# B&R Automation Studio project Ampel (part 5)

```cpp
#if HFSM2_PLANS_AVAILABLE()
		HFSM2_CONSTEXPR(14)	TaskStatus	wideUpdatePlans		 ( FullControl& control												   )		noexcept;
#endif

		HFSM2_CONSTEXPR(14)	bool		wideForwardExitGuard (GuardControl& control,						const ProngCBits prongs)		noexcept;
		HFSM2_CONSTEXPR(14)	bool		wideForwardExitGuard (GuardControl& control												   )		noexcept;
		HFSM2_CONSTEXPR(14)	bool		wideExitGuard		 (GuardControl& control												   )		noexcept;

		HFSM2_CONSTEXPR(14)	void		wideExit			 ( PlanControl& control												   )		noexcept;

		HFSM2_CONSTEXPR(14)	void		wideForwardActive	 (	   Control& control, const Request request, const ProngCBits prongs)		noexcept;
		HFSM2_CONSTEXPR(14)	void		wideForwardRequest	 (	   Control& control, const Request request						   )		noexcept;

		HFSM2_CONSTEXPR(14)	void		wideRequestChange	 (	   Control& control, const Request request						   )		noexcept;
		HFSM2_CONSTEXPR(14)	void		wideRequestRestart	 (	   Control& control, const Request request						   )		noexcept;
		HFSM2_CONSTEXPR(14)	void		wideRequestResume	 (	   Control& control, const Request request						   )		noexcept;
		HFSM2_CONSTEXPR(14)	void		wideRequestSelect	 (	   Control& control, const Request request						   )		noexcept;

#if HFSM2_UTILITY_THEORY_AVAILABLE()
		HFSM2_CONSTEXPR(14)	void		wideRequestUtilize	 (	   Control& control, const Request request						   )		noexcept;
		HFSM2_CONSTEXPR(14)	void		wideRequestRandomize (	   Control& control, const Request request						   )		noexcept;

		HFSM2_CONSTEXPR(14)	Utility		wideReportChange	 (	   Control& control												   )		noexcept;
		HFSM2_CONSTEXPR(14)	Utility		wideReportUtilize	 (	   Control& control												   )		noexcept;
		HFSM2_CONSTEXPR(14)	Utility		wideReportRandomize  (	   Control& control												   )		noexcept;
#endif

		HFSM2_CONSTEXPR(14)	void		wideChangeToRequested( PlanControl& control												   )		noexcept;

#if HFSM2_SERIALIZATION_AVAILABLE()
		using WriteStream	= typename Args::WriteStream;
		using ReadStream	= typename Args::ReadStream;

		HFSM2_CONSTEXPR(14)	void		wideSaveActive		  (const Registry& registry, WriteStream& stream)  const noexcept;
		HFSM2_CONSTEXPR(14)	void		wideSaveResumable	  (const Registry& registry, WriteStream& stream)  const noexcept;

		HFSM2_CONSTEXPR(14)	void		wideLoadRequested	  (		 Registry& registry,  ReadStream& stream)  const noexcept;
		HFSM2_CONSTEXPR(14)	void		wideLoadResumable	  (		 Registry& registry,  ReadStream& stream)  const noexcept;
#endif

#if HFSM2_STRUCTURE_REPORT_AVAILABLE()
		using StructureStateInfos = typename Args::StructureStateInfos;

		static constexpr Long NAME_COUNT	 = Initial::NAME_COUNT  + Remaining::NAME_COUNT;

		HFSM2_CONSTEXPR(14)	void wideGetNames(const Long parent,
		const Short depth,
		StructureStateInfos& stateInfos)	  const noexcept;
#endif

	};

}
}

namespace hfsm2 {
	namespace detail {

		template <typename TN_, typename TA_, Prong NP_, typename TI_, typename... TR_>
		HFSM2_CONSTEXPR(14)
		void
		OS_<TN_, TA_, NP_, TI_, TR_...>::wideRegister(Registry& registry,
		const ForkID forkId) noexcept
		{
		Initial	 ::deepRegister(registry, Parent{forkId, PRONG_INDEX});
		Remaining::wideRegister(registry,		 forkId				 );
	}

	template <typename TN_, typename TA_, Prong NP_, typename TI_, typename... TR_>
	HFSM2_CONSTEXPR(14)
	bool
	OS_<TN_, TA_, NP_, TI_, TR_...>::wideForwardEntryGuard(GuardControl& control,
	const ProngCBits prongs) noexcept
	{
	const bool i = prongs.get(PRONG_INDEX) ?
		Initial	::deepForwardEntryGuard(control		   ) : false;

	const bool r = Remaining::wideForwardEntryGuard(control, prongs);

	return i || r;
}

template <typename TN_, typename TA_, Prong NP_, typename TI_, typename... TR_>
HFSM2_CONSTEXPR(14)
bool
OS_<TN_, TA_, NP_, TI_, TR_...>::wideForwardEntryGuard(GuardControl& control) noexcept {
const bool i = Initial	::deepForwardEntryGuard(control);
const bool r = Remaining::wideForwardEntryGuard(control);

return i || r;
}

template <typename TN_, typename TA_, Prong NP_, typename TI_, typename... TR_>
HFSM2_CONSTEXPR(14)
bool
OS_<TN_, TA_, NP_, TI_, TR_...>::wideEntryGuard(GuardControl& control) noexcept {
const bool i = Initial	::deepEntryGuard(control);
const bool r = Remaining::wideEntryGuard(control);

return i || r;
}

template <typename TN_, typename TA_, Prong NP_, typename TI_, typename... TR_>
HFSM2_CONSTEXPR(14)
void
OS_<TN_, TA_, NP_, TI_, TR_...>::wideEnter(PlanControl& control) noexcept {
	Initial	 ::deepEnter(control);
	Remaining::wideEnter(control);
}

template <typename TN_, typename TA_, Prong NP_, typename TI_, typename... TR_>
HFSM2_CONSTEXPR(14)
void
OS_<TN_, TA_, NP_, TI_, TR_...>::wideReenter(PlanControl& control) noexcept {
	Initial	 ::deepReenter(control);
	Remaining::wideReenter(control);
}

template <typename TN_, typename TA_, Prong NP_, typename TI_, typename... TR_>
HFSM2_CONSTEXPR(14)
TaskStatus
OS_<TN_, TA_, NP_, TI_, TR_...>::widePreUpdate(FullControl& control) noexcept {
TaskStatus status;
	status |= Initial  ::deepPreUpdate(control);
	status |= Remaining::widePreUpdate(control);

return status;
}

template <typename TN_, typename TA_, Prong NP_, typename TI_, typename... TR_>
HFSM2_CONSTEXPR(14)
TaskStatus
OS_<TN_, TA_, NP_, TI_, TR_...>::wideUpdate(FullControl& control) noexcept {
TaskStatus status;
	status |= Initial  ::deepUpdate(control);
	status |= Remaining::wideUpdate(control);

return status;
}

template <typename TN_, typename TA_, Prong NP_, typename TI_, typename... TR_>
HFSM2_CONSTEXPR(14)
TaskStatus
OS_<TN_, TA_, NP_, TI_, TR_...>::widePostUpdate(FullControl& control) noexcept {
TaskStatus status;
	status |= Initial  ::deepPostUpdate(control);
	status |= Remaining::widePostUpdate(control);

return status;
}

template <typename TN_, typename TA_, Prong NP_, typename TI_, typename... TR_>
template <typename TEvent>
HFSM2_CONSTEXPR(14)
TaskStatus
OS_<TN_, TA_, NP_, TI_, TR_...>::widePreReact(EventControl& control,
											  const TEvent& event) noexcept
{
TaskStatus status;
	status |= Initial  ::deepPreReact(control, event);
	status |= Remaining::widePreReact(control, event);

return status;
}

template <typename TN_, typename TA_, Prong NP_, typename TI_, typename... TR_>
template <typename TEvent>
HFSM2_CONSTEXPR(14)
TaskStatus
OS_<TN_, TA_, NP_, TI_, TR_...>::wideReact(EventControl& control,
										   const TEvent& event) noexcept
{
TaskStatus status;
	status |= Initial  ::deepReact(control, event);
	status |= Remaining::wideReact(control, event);

return status;
}

template <typename TN_, typename TA_, Prong NP_, typename TI_, typename... TR_>
template <typename TEvent>
HFSM2_CONSTEXPR(14)
TaskStatus
OS_<TN_, TA_, NP_, TI_, TR_...>::widePostReact(EventControl& control,
											   const TEvent& event) noexcept
{
TaskStatus status;
	status |= Initial  ::deepPostReact(control, event);
	status |= Remaining::widePostReact(control, event);

return status;
}

template <typename TN_, typename TA_, Prong NP_, typename TI_, typename... TR_>
template <typename TEvent>
HFSM2_CONSTEXPR(14)
void
OS_<TN_, TA_, NP_, TI_, TR_...>::wideQuery(ConstControl& control,
										   TEvent& event) const noexcept
{
	Initial  ::deepQuery(control, event);
	Remaining::wideQuery(control, event);
}

#if HFSM2_PLANS_AVAILABLE()

template <typename TN_, typename TA_, Prong NP_, typename TI_, typename... TR_>
HFSM2_CONSTEXPR(14)
TaskStatus
OS_<TN_, TA_, NP_, TI_, TR_...>::wideUpdatePlans(FullControl& control) noexcept {
TaskStatus status;
	status |= Initial  ::deepUpdatePlans(control);
	status |= Remaining::wideUpdatePlans(control);

return status;
}

#endif

template <typename TN_, typename TA_, Prong NP_, typename TI_, typename... TR_>
HFSM2_CONSTEXPR(14)
bool
OS_<TN_, TA_, NP_, TI_, TR_...>::wideForwardExitGuard(GuardControl& control,
													  const ProngCBits prongs) noexcept
{
const bool i = prongs.get(PRONG_INDEX) ?
	Initial	::deepForwardExitGuard(control		  ) : false;

const bool r = Remaining::wideForwardExitGuard(control, prongs);

return i || r;
}

template <typename TN_, typename TA_, Prong NP_, typename TI_, typename... TR_>
HFSM2_CONSTEXPR(14)
bool
OS_<TN_, TA_, NP_, TI_, TR_...>::wideForwardExitGuard(GuardControl& control) noexcept {
const bool i = Initial	::deepForwardExitGuard(control);
const bool r = Remaining::wideForwardExitGuard(control);

return i || r;
}

template <typename TN_, typename TA_, Prong NP_, typename TI_, typename... TR_>
HFSM2_CONSTEXPR(14)
bool
OS_<TN_, TA_, NP_, TI_, TR_...>::wideExitGuard(GuardControl& control) noexcept {
const bool i = Initial	::deepExitGuard(control);
const bool r = Remaining::wideExitGuard(control);

return i || r;
}

template <typename TN_, typename TA_, Prong NP_, typename TI_, typename... TR_>
HFSM2_CONSTEXPR(14)
void
OS_<TN_, TA_, NP_, TI_, TR_...>::wideExit(PlanControl& control) noexcept {
	Initial	 ::deepExit(control);
	Remaining::wideExit(control);
}

template <typename TN_, typename TA_, Prong NP_, typename TI_, typename... TR_>
HFSM2_CONSTEXPR(14)
void
OS_<TN_, TA_, NP_, TI_, TR_...>::wideForwardActive(Control& control,
												   const Request request,
												   const ProngCBits prongs) noexcept
{
	if (prongs.get(PRONG_INDEX))
		Initial::deepForwardActive(control, request		   );

	Remaining  ::wideForwardActive(control, request, prongs);
}

template <typename TN_, typename TA_, Prong NP_, typename TI_, typename... TR_>
HFSM2_CONSTEXPR(14)
void
OS_<TN_, TA_, NP_, TI_, TR_...>::wideForwardRequest(Control& control,
													const Request request) noexcept
{
	Initial	 ::deepForwardRequest(control, request);
	Remaining::wideForwardRequest(control, request);
}

template <typename TN_, typename TA_, Prong NP_, typename TI_, typename... TR_>
HFSM2_CONSTEXPR(14)
void
OS_<TN_, TA_, NP_, TI_, TR_...>::wideRequestChange(Control& control,
												   const Request request) noexcept
{
	Initial	 ::deepRequestChange(control, request);
	Remaining::wideRequestChange(control, request);
}

template <typename TN_, typename TA_, Prong NP_, typename TI_, typename... TR_>
HFSM2_CONSTEXPR(14)
void
OS_<TN_, TA_, NP_, TI_, TR_...>::wideRequestRestart(Control& control,
													const Request request) noexcept
{
	Initial	 ::deepRequestRestart(control, request);
	Remaining::wideRequestRestart(control, request);
}

template <typename TN_, typename TA_, Prong NP_, typename TI_, typename... TR_>
HFSM2_CONSTEXPR(14)
void
OS_<TN_, TA_, NP_, TI_, TR_...>::wideRequestResume(Control& control,
												   const Request request) noexcept
{
	Initial	 ::deepRequestResume(control, request);
	Remaining::wideRequestResume(control, request);
}

template <typename TN_, typename TA_, Prong NP_, typename TI_, typename... TR_>
HFSM2_CONSTEXPR(14)
void
OS_<TN_, TA_, NP_, TI_, TR_...>::wideRequestSelect(Control& control,
												   const Request request) noexcept
{
	Initial	 ::deepRequestSelect(control, request);
	Remaining::wideRequestSelect(control, request);
}

#if HFSM2_UTILITY_THEORY_AVAILABLE()

template <typename TN_, typename TA_, Prong NP_, typename TI_, typename... TR_>
HFSM2_CONSTEXPR(14)
void
OS_<TN_, TA_, NP_, TI_, TR_...>::wideRequestUtilize(Control& control,
													const Request request) noexcept
{
	Initial	 ::deepRequestUtilize(control, request);
	Remaining::wideRequestUtilize(control, request);
}

template <typename TN_, typename TA_, Prong NP_, typename TI_, typename... TR_>
HFSM2_CONSTEXPR(14)
void
OS_<TN_, TA_, NP_, TI_, TR_...>::wideRequestRandomize(Control& control,
													  const Request request) noexcept
{
	Initial	 ::deepRequestRandomize(control, request);
	Remaining::wideRequestRandomize(control, request);
}

template <typename TN_, typename TA_, Prong NP_, typename TI_, typename... TR_>
HFSM2_CONSTEXPR(14)
typename TA_::Utility
OS_<TN_, TA_, NP_, TI_, TR_...>::wideReportChange(Control& control) noexcept {
const UP	  i = Initial  ::deepReportChange(control);
const Utility r = Remaining::wideReportChange(control);

return i.utility + r;
}

template <typename TN_, typename TA_, Prong NP_, typename TI_, typename... TR_>
HFSM2_CONSTEXPR(14)
typename TA_::Utility
OS_<TN_, TA_, NP_, TI_, TR_...>::wideReportUtilize(Control& control) noexcept {
const UP	  i = Initial  ::deepReportUtilize(control);
const Utility r = Remaining::wideReportUtilize(control);

return i.utility + r;
}

template <typename TN_, typename TA_, Prong NP_, typename TI_, typename... TR_>
HFSM2_CONSTEXPR(14)
typename TA_::Utility
OS_<TN_, TA_, NP_, TI_, TR_...>::wideReportRandomize(Control& control) noexcept {
const Utility i = Initial  ::deepReportRandomize(control);
const Utility r = Remaining::wideReportRandomize(control);

return i + r;
}

#endif

template <typename TN_, typename TA_, Prong NP_, typename TI_, typename... TR_>
HFSM2_CONSTEXPR(14)
void
OS_<TN_, TA_, NP_, TI_, TR_...>::wideChangeToRequested(PlanControl& control) noexcept {
	Initial	 ::deepChangeToRequested(control);
	Remaining::wideChangeToRequested(control);
}

#if HFSM2_SERIALIZATION_AVAILABLE()

template <typename TN_, typename TA_, Prong NP_, typename TI_, typename... TR_>
HFSM2_CONSTEXPR(14)
void
OS_<TN_, TA_, NP_, TI_, TR_...>::wideSaveActive(const Registry& registry,
												WriteStream& stream) const noexcept
{
	Initial	 ::deepSaveActive(registry, stream);
	Remaining::wideSaveActive(registry, stream);
}

template <typename TN_, typename TA_, Prong NP_, typename TI_, typename... TR_>
HFSM2_CONSTEXPR(14)
void
OS_<TN_, TA_, NP_, TI_, TR_...>::wideSaveResumable(const Registry& registry,
												   WriteStream& stream) const noexcept
{
	Initial	 ::deepSaveResumable(registry, stream);
	Remaining::wideSaveResumable(registry, stream);
}

template <typename TN_, typename TA_, Prong NP_, typename TI_, typename... TR_>
HFSM2_CONSTEXPR(14)
void
OS_<TN_, TA_, NP_, TI_, TR_...>::wideLoadRequested(Registry& registry,
												   ReadStream& stream) const noexcept
{
	Initial	 ::deepLoadRequested(registry, stream);
	Remaining::wideLoadRequested(registry, stream);
}

template <typename TN_, typename TA_, Prong NP_, typename TI_, typename... TR_>
HFSM2_CONSTEXPR(14)
void
OS_<TN_, TA_, NP_, TI_, TR_...>::wideLoadResumable(Registry& registry,
												   ReadStream& stream) const noexcept
{
	Initial	 ::deepLoadResumable(registry, stream);
	Remaining::wideLoadResumable(registry, stream);
}

#endif

#if HFSM2_STRUCTURE_REPORT_AVAILABLE()

template <typename TN_, typename TA_, Prong NP_, typename TI_, typename... TR_>
HFSM2_CONSTEXPR(14)
void
OS_<TN_, TA_, NP_, TI_, TR_...>::wideGetNames(const Long parent,
											  const Short depth,
											  StructureStateInfos& stateInfos) const noexcept
{
	Initial	 ::deepGetNames(parent, RegionType::ORTHOGONAL, depth, stateInfos);
	Remaining::wideGetNames(parent						  , depth, stateInfos);
}

#endif

}
}

namespace hfsm2 {
	namespace detail {

		template <
		typename TIndices
		, typename TArgs
		, Prong NProng
		, typename TInitial
		>
		struct HFSM2_EMPTY_BASES OS_<
			TIndices
			, TArgs
			, NProng
			, TInitial
			>
			:					 InitialOS<
			TIndices
			, TArgs
			, TInitial
			>
			{
			using Indices		= TIndices;
			static constexpr StateID INITIAL_ID	 = Indices::STATE_ID;
			static constexpr Short	 COMPO_INDEX = Indices::COMPO_INDEX;
			static constexpr Short	 ORTHO_INDEX = Indices::ORTHO_INDEX;
			static constexpr Short	 ORTHO_UNIT	 = Indices::ORTHO_UNIT;

			static constexpr Prong	 PRONG_INDEX = NProng;

			using Args			= TArgs;

#if HFSM2_UTILITY_THEORY_AVAILABLE()
			using Rank			= typename Args::Rank;
			using Utility		= typename Args::Utility;
			using UP			= typename Args::UP;
#endif

			using Registry		= RegistryT<Args>;
			using StateParents	= typename Registry::StateParents;
			using OrthoForks	= typename Registry::OrthoForks;
			using ProngBits		= typename OrthoForks::Bits;
			using ProngCBits	= typename OrthoForks::CBits;

			using ConstControl	= ConstControlT<Args>;
			using Control		= ControlT	   <Args>;
			using PlanControl	= PlanControlT <Args>;
			using FullControl	= FullControlT <Args>;
			using GuardControl	= GuardControlT<Args>;
			using EventControl	= EventControlT<Args>;

			using Initial		= InitialOS<
				TIndices,
				TArgs,
				TInitial
				>;

			HFSM2_CONSTEXPR(14)	void		wideRegister		 (Registry& registry, const ForkID forkId)										noexcept;

			HFSM2_CONSTEXPR(14)	bool		wideForwardEntryGuard(GuardControl& control,						const ProngCBits prongs)		noexcept;
			HFSM2_CONSTEXPR(14)	bool		wideForwardEntryGuard(GuardControl& control												   )		noexcept;
			HFSM2_CONSTEXPR(14)	bool		wideEntryGuard		 (GuardControl& control												   )		noexcept;

			HFSM2_CONSTEXPR(14)	void		wideEnter			 ( PlanControl& control												   )		noexcept;
			HFSM2_CONSTEXPR(14)	void		wideReenter			 ( PlanControl& control												   )		noexcept;

			HFSM2_CONSTEXPR(14)	TaskStatus	widePreUpdate		 ( FullControl& control												   )		noexcept;
			HFSM2_CONSTEXPR(14)	TaskStatus	wideUpdate			 ( FullControl& control												   )		noexcept;
			HFSM2_CONSTEXPR(14)	TaskStatus	widePostUpdate		 ( FullControl& control												   )		noexcept;

			template <typename TEvent>
			HFSM2_CONSTEXPR(14)	TaskStatus	widePreReact		 (EventControl& control, const TEvent& event						   )		noexcept;

			template <typename TEvent>
			HFSM2_CONSTEXPR(14)	TaskStatus	wideReact			 (EventControl& control, const TEvent& event						   )		noexcept;

			template <typename TEvent>
			HFSM2_CONSTEXPR(14)	TaskStatus	widePostReact		 (EventControl& control, const TEvent& event						   )		noexcept;

			template <typename TEvent>
			HFSM2_CONSTEXPR(14)	void		wideQuery			 (ConstControl& control,	   TEvent& event						   )  const noexcept;

#if HFSM2_PLANS_AVAILABLE()
			HFSM2_CONSTEXPR(14)	TaskStatus	wideUpdatePlans		 ( FullControl& control												   )		noexcept;
#endif

			HFSM2_CONSTEXPR(14)	bool		wideForwardExitGuard (GuardControl& control,						const ProngCBits prongs)		noexcept;
			HFSM2_CONSTEXPR(14)	bool		wideForwardExitGuard (GuardControl& control												   )		noexcept;
			HFSM2_CONSTEXPR(14)	bool		wideExitGuard		 (GuardControl& control												   )		noexcept;

			HFSM2_CONSTEXPR(14)	void		wideExit			 ( PlanControl& control												   )		noexcept;

			HFSM2_CONSTEXPR(14)	void		wideForwardActive	 (	   Control& control, const Request request, const ProngCBits prongs)		noexcept;
			HFSM2_CONSTEXPR(14)	void		wideForwardRequest	 (	   Control& control, const Request request						   )		noexcept;

			HFSM2_CONSTEXPR(14)	void		wideRequestChange	 (	   Control& control, const Request request						   )		noexcept;
			HFSM2_CONSTEXPR(14)	void		wideRequestRestart	 (	   Control& control, const Request request						   )		noexcept;
			HFSM2_CONSTEXPR(14)	void		wideRequestResume	 (	   Control& control, const Request request						   )		noexcept;
			HFSM2_CONSTEXPR(14)	void		wideRequestSelect	 (	   Control& control, const Request request						   )		noexcept;

#if HFSM2_UTILITY_THEORY_AVAILABLE()
			HFSM2_CONSTEXPR(14)	void		wideRequestUtilize	 (	   Control& control, const Request request						   )		noexcept;
			HFSM2_CONSTEXPR(14)	void		wideRequestRandomize (	   Control& control, const Request request						   )		noexcept;

			HFSM2_CONSTEXPR(14)	Utility		wideReportChange	 (	   Control& control												   )		noexcept;
			HFSM2_CONSTEXPR(14)	Utility		wideReportUtilize	 (	   Control& control												   )		noexcept;
			HFSM2_CONSTEXPR(14)	Utility		wideReportRandomize  (	   Control& control												   )		noexcept;
#endif

			HFSM2_CONSTEXPR(14)	void		wideChangeToRequested( PlanControl& control												   )		noexcept;

#if HFSM2_SERIALIZATION_AVAILABLE()
			using WriteStream	= typename Args::WriteStream;
			using ReadStream	= typename Args::ReadStream;

			HFSM2_CONSTEXPR(14)	void		wideSaveActive		  (const Registry& registry, WriteStream& stream)  const noexcept;
			HFSM2_CONSTEXPR(14)	void		wideSaveResumable	  (const Registry& registry, WriteStream& stream)  const noexcept;

			HFSM2_CONSTEXPR(14)	void		wideLoadRequested	  (		 Registry& registry,  ReadStream& stream)  const noexcept;
			HFSM2_CONSTEXPR(14)	void		wideLoadResumable	  (		 Registry& registry,  ReadStream& stream)  const noexcept;
#endif

#if HFSM2_STRUCTURE_REPORT_AVAILABLE()
			using StructureStateInfos = typename Args::StructureStateInfos;

			static constexpr Long NAME_COUNT	 = Initial::NAME_COUNT;

			HFSM2_CONSTEXPR(14)	void wideGetNames(const Long parent,
			const Short depth,
			StructureStateInfos& stateInfos)							  const noexcept;
#endif

		};

	}
}

namespace hfsm2 {
	namespace detail {

		template <typename TN_, typename TA_, Prong NP_, typename TI_>
		HFSM2_CONSTEXPR(14)
		void
		OS_<TN_, TA_, NP_, TI_>::wideRegister(Registry& registry,
		const ForkID forkId) noexcept
		{
		Initial::deepRegister(registry, Parent{forkId, PRONG_INDEX});
	}

	template <typename TN_, typename TA_, Prong NP_, typename TI_>
	HFSM2_CONSTEXPR(14)
	bool
	OS_<TN_, TA_, NP_, TI_>::wideForwardEntryGuard(GuardControl& control,
	const ProngCBits prongs) noexcept
	{
	return prongs.get(PRONG_INDEX) ?
	Initial::deepForwardEntryGuard(control) : false;
}

template <typename TN_, typename TA_, Prong NP_, typename TI_>
HFSM2_CONSTEXPR(14)
bool
OS_<TN_, TA_, NP_, TI_>::wideForwardEntryGuard(GuardControl& control) noexcept {
	return Initial::deepForwardEntryGuard(control);
}

template <typename TN_, typename TA_, Prong NP_, typename TI_>
HFSM2_CONSTEXPR(14)
bool
OS_<TN_, TA_, NP_, TI_>::wideEntryGuard(GuardControl& control) noexcept {
	return Initial::deepEntryGuard(control);
}

template <typename TN_, typename TA_, Prong NP_, typename TI_>
HFSM2_CONSTEXPR(14)
void
OS_<TN_, TA_, NP_, TI_>::wideEnter(PlanControl& control) noexcept {
	Initial::deepEnter(control);
}

template <typename TN_, typename TA_, Prong NP_, typename TI_>
HFSM2_CONSTEXPR(14)
void
OS_<TN_, TA_, NP_, TI_>::wideReenter(PlanControl& control) noexcept {
	Initial::deepReenter(control);
}

template <typename TN_, typename TA_, Prong NP_, typename TI_>
HFSM2_CONSTEXPR(14)
TaskStatus
OS_<TN_, TA_, NP_, TI_>::widePreUpdate(FullControl& control) noexcept {
	return Initial::deepPreUpdate(control);
}

template <typename TN_, typename TA_, Prong NP_, typename TI_>
HFSM2_CONSTEXPR(14)
TaskStatus
OS_<TN_, TA_, NP_, TI_>::wideUpdate(FullControl& control) noexcept {
	return Initial::deepUpdate(control);
}

template <typename TN_, typename TA_, Prong NP_, typename TI_>
HFSM2_CONSTEXPR(14)
TaskStatus
OS_<TN_, TA_, NP_, TI_>::widePostUpdate(FullControl& control) noexcept {
	return Initial::deepPostUpdate(control);
}

template <typename TN_, typename TA_, Prong NP_, typename TI_>
template <typename TEvent>
HFSM2_CONSTEXPR(14)
TaskStatus
OS_<TN_, TA_, NP_, TI_>::widePreReact(EventControl& control,
									  const TEvent& event) noexcept
{
	return Initial::deepPreReact(control, event);
}

template <typename TN_, typename TA_, Prong NP_, typename TI_>
template <typename TEvent>
HFSM2_CONSTEXPR(14)
TaskStatus
OS_<TN_, TA_, NP_, TI_>::wideReact(EventControl& control,
								   const TEvent& event) noexcept
{
	return Initial::deepReact(control, event);
}

template <typename TN_, typename TA_, Prong NP_, typename TI_>
template <typename TEvent>
HFSM2_CONSTEXPR(14)
TaskStatus
OS_<TN_, TA_, NP_, TI_>::widePostReact(EventControl& control,
									   const TEvent& event) noexcept
{
	return Initial::deepPostReact(control, event);
}

template <typename TN_, typename TA_, Prong NP_, typename TI_>
template <typename TEvent>
HFSM2_CONSTEXPR(14)
void
	OS_<TN_, TA_, NP_, TI_>::wideQuery(ConstControl& control,
	TEvent& event) const noexcept
{
	Initial::deepQuery(control, event);
}

#if HFSM2_PLANS_AVAILABLE()

template <typename TN_, typename TA_, Prong NP_, typename TI_>
HFSM2_CONSTEXPR(14)
TaskStatus
OS_<TN_, TA_, NP_, TI_>::wideUpdatePlans(FullControl& control) noexcept {
	return Initial::deepUpdatePlans(control);
}

#endif

template <typename TN_, typename TA_, Prong NP_, typename TI_>
HFSM2_CONSTEXPR(14)
bool
OS_<TN_, TA_, NP_, TI_>::wideForwardExitGuard(GuardControl& control,
											  const ProngCBits prongs) noexcept
{
	return prongs.get(PRONG_INDEX) ?
		Initial::deepForwardExitGuard(control) : false;
}

template <typename TN_, typename TA_, Prong NP_, typename TI_>
HFSM2_CONSTEXPR(14)
bool
OS_<TN_, TA_, NP_, TI_>::wideForwardExitGuard(GuardControl& control) noexcept {
	return Initial::deepForwardExitGuard(control);
}

template <typename TN_, typename TA_, Prong NP_, typename TI_>
HFSM2_CONSTEXPR(14)
bool
OS_<TN_, TA_, NP_, TI_>::wideExitGuard(GuardControl& control) noexcept {
	return Initial::deepExitGuard(control);
}

template <typename TN_, typename TA_, Prong NP_, typename TI_>
HFSM2_CONSTEXPR(14)
void
OS_<TN_, TA_, NP_, TI_>::wideExit(PlanControl& control) noexcept {
	Initial::deepExit(control);
}

template <typename TN_, typename TA_, Prong NP_, typename TI_>
HFSM2_CONSTEXPR(14)
void
OS_<TN_, TA_, NP_, TI_>::wideForwardActive(Control& control,
										   const Request request,
										   const ProngCBits prongs) noexcept
{
	if (prongs.get(PRONG_INDEX))
		Initial::deepForwardActive(control, request);
}

template <typename TN_, typename TA_, Prong NP_, typename TI_>
HFSM2_CONSTEXPR(14)
void
OS_<TN_, TA_, NP_, TI_>::wideForwardRequest(Control& control,
											const Request request) noexcept
{
	Initial::deepForwardRequest(control, request);
}

template <typename TN_, typename TA_, Prong NP_, typename TI_>
HFSM2_CONSTEXPR(14)
void
OS_<TN_, TA_, NP_, TI_>::wideRequestChange(Control& control,
										   const Request request) noexcept
{
	Initial::deepRequestChange(control, request);
}

template <typename TN_, typename TA_, Prong NP_, typename TI_>
HFSM2_CONSTEXPR(14)
void
OS_<TN_, TA_, NP_, TI_>::wideRequestRestart(Control& control,
											const Request request) noexcept
{
	Initial::deepRequestRestart(control, request);
}

template <typename TN_, typename TA_, Prong NP_, typename TI_>
HFSM2_CONSTEXPR(14)
void
OS_<TN_, TA_, NP_, TI_>::wideRequestResume(Control& control,
										   const Request request) noexcept
{
	Initial::deepRequestResume(control, request);
}

template <typename TN_, typename TA_, Prong NP_, typename TI_>
HFSM2_CONSTEXPR(14)
void
OS_<TN_, TA_, NP_, TI_>::wideRequestSelect(Control& control,
										   const Request request) noexcept
{
	Initial::deepRequestSelect(control, request);
}

#if HFSM2_UTILITY_THEORY_AVAILABLE()

template <typename TN_, typename TA_, Prong NP_, typename TI_>
HFSM2_CONSTEXPR(14)
void
OS_<TN_, TA_, NP_, TI_>::wideRequestUtilize(Control& control,
											const Request request) noexcept
{
	Initial::deepRequestUtilize(control, request);
}

template <typename TN_, typename TA_, Prong NP_, typename TI_>
HFSM2_CONSTEXPR(14)
void
OS_<TN_, TA_, NP_, TI_>::wideRequestRandomize(Control& control,
											  const Request request) noexcept
{
	Initial::deepRequestRandomize(control, request);
}

template <typename TN_, typename TA_, Prong NP_, typename TI_>
HFSM2_CONSTEXPR(14)
typename TA_::Utility
OS_<TN_, TA_, NP_, TI_>::wideReportChange(Control& control) noexcept {
const UP i = Initial::deepReportChange(control);

return i.utility;
}

template <typename TN_, typename TA_, Prong NP_, typename TI_>
HFSM2_CONSTEXPR(14)
typename TA_::Utility
OS_<TN_, TA_, NP_, TI_>::wideReportUtilize(Control& control) noexcept {
const UP i = Initial::deepReportUtilize(control);

return i.utility;
}

template <typename TN_, typename TA_, Prong NP_, typename TI_>
HFSM2_CONSTEXPR(14)
typename TA_::Utility
OS_<TN_, TA_, NP_, TI_>::wideReportRandomize(Control& control) noexcept {
	return Initial::deepReportRandomize(control);
}

#endif

template <typename TN_, typename TA_, Prong NP_, typename TI_>
HFSM2_CONSTEXPR(14)
void
OS_<TN_, TA_, NP_, TI_>::wideChangeToRequested(PlanControl& control) noexcept {
	Initial::deepChangeToRequested(control);
}

#if HFSM2_SERIALIZATION_AVAILABLE()

template <typename TN_, typename TA_, Prong NP_, typename TI_>
HFSM2_CONSTEXPR(14)
void
	OS_<TN_, TA_, NP_, TI_>::wideSaveActive(const Registry& registry,
	WriteStream& stream) const noexcept
{
	Initial::deepSaveActive(registry, stream);
}

template <typename TN_, typename TA_, Prong NP_, typename TI_>
HFSM2_CONSTEXPR(14)
void
	OS_<TN_, TA_, NP_, TI_>::wideSaveResumable(const Registry& registry,
	WriteStream& stream) const noexcept
{
	Initial::deepSaveResumable(registry, stream);
}

template <typename TN_, typename TA_, Prong NP_, typename TI_>
HFSM2_CONSTEXPR(14)
void
	OS_<TN_, TA_, NP_, TI_>::wideLoadRequested(Registry& registry,
	ReadStream& stream) const noexcept
{
	Initial::deepLoadRequested(registry, stream);
}

template <typename TN_, typename TA_, Prong NP_, typename TI_>
HFSM2_CONSTEXPR(14)
void
	OS_<TN_, TA_, NP_, TI_>::wideLoadResumable(Registry& registry,
	ReadStream& stream) const noexcept
{
	Initial::deepLoadResumable(registry, stream);
}

#endif

#if HFSM2_STRUCTURE_REPORT_AVAILABLE()

template <typename TN_, typename TA_, Prong NP_, typename TI_>
HFSM2_CONSTEXPR(14)
void
	OS_<TN_, TA_, NP_, TI_>::wideGetNames(const Long parent,
	const Short depth,
	StructureStateInfos& stateInfos) const noexcept
{
	Initial::deepGetNames(parent, RegionType::ORTHOGONAL, depth, stateInfos);
}

#endif

}
}

namespace hfsm2 {
	namespace detail {

		template <
		typename TIndices
		, typename TArgs
		, typename THead
		, typename... TSubStates
		>
		struct HFSM2_EMPTY_BASES O_
		: S_<TIndices, TArgs, THead>
		, OS_<
		I_<
		TIndices::STATE_ID + 1
		, TIndices::COMPO_INDEX
		, TIndices::ORTHO_INDEX + 1
		, TIndices::ORTHO_UNIT + contain(OI_<THead, TSubStates...>::WIDTH, 8)
		>
		, TArgs
		, 0
		, TSubStates...
		>
		{
		using Indices		= TIndices;
		static constexpr StateID  HEAD_ID	  = Indices::STATE_ID;
		static constexpr Short	  COMPO_INDEX = Indices::COMPO_INDEX;
		static constexpr Short	  ORTHO_INDEX = Indices::ORTHO_INDEX;
		static constexpr Short	  ORTHO_UNIT  = Indices::ORTHO_UNIT;

		static constexpr RegionID REGION_ID	  = COMPO_INDEX + ORTHO_INDEX;
		static constexpr ForkID	  ORTHO_ID	  = static_cast<ForkID>(-ORTHO_INDEX - 1);

		using Args			= TArgs;

#if HFSM2_UTILITY_THEORY_AVAILABLE()
		using Rank			= typename Args::Rank;
		using Utility		= typename Args::Utility;
		using UP			= typename Args::UP;
#endif

		using StateList		= typename Args::StateList;
		using RegionList	= typename Args::RegionList;

		using ReactOrder	= typename Args::ReactOrder;

		using Registry		= RegistryT<Args>;
		using StateParents	= typename Registry::StateParents;
		using OrthoForks	= typename Registry::OrthoForks;
		using ProngBits		= typename OrthoForks::Bits;
		using ProngCBits	= typename OrthoForks::CBits;

		using ConstControl	= ConstControlT<Args>;
		using ScopedCRegion	= typename ConstControl::Region;

		using Control		= ControlT	   <Args>;
		using ScopedOrigin	= typename Control::Origin;

		using PlanControl	= PlanControlT <Args>;
		using FullControl	= FullControlT <Args>;
		using ControlLock	= typename FullControl::Lock;
		using ScopedRegion	= typename PlanControl::Region;

		using GuardControl	= GuardControlT<Args>;
		using EventControl	= EventControlT<Args>;

		using Head			= THead;
		using HeadState		= S_<Indices, Args, Head>;

		using Info			= OI_<Head, TSubStates...>;
		static constexpr Short WIDTH		= Info::WIDTH;
		static constexpr Long  REGION_SIZE	= Info::STATE_COUNT;
		static constexpr Short ORTHO_UNITS	= Info::ORTHO_UNITS;

		using SubStates		= OS_<
			I_<
			HEAD_ID + 1,
			COMPO_INDEX,
			ORTHO_INDEX + 1,
			ORTHO_UNIT + contain(WIDTH, 8)
			>,
		Args,
		0,
		TSubStates...
		>;

		using PreReactWrapper	= PreReactWrapperT <O_, ReactOrder>;
		using ReactWrapper		= ReactWrapperT	   <O_, ReactOrder>;
		using PostReactWrapper	= PostReactWrapperT<O_, ReactOrder>;
		using QueryWrapper		= QueryWrapperT	   <O_, ReactOrder>;

	HFSM2_CONSTEXPR(11)	static ProngBits  orthoRequested (		Registry& registry)		noexcept	{ return			   registry.orthoRequested.template  bits<ORTHO_UNIT, WIDTH>();	}
HFSM2_CONSTEXPR(11)	static ProngCBits orthoRequested (const Registry& registry)		noexcept	{ return			   registry.orthoRequested.template cbits<ORTHO_UNIT, WIDTH>();	}

	HFSM2_CONSTEXPR(11)	static ProngBits  orthoRequested (		Control& control )		noexcept	{ return control._core.registry.orthoRequested.template  bits<ORTHO_UNIT, WIDTH>();	}
	HFSM2_CONSTEXPR(11)	static ProngCBits orthoRequested (const	Control& control )		noexcept	{ return control._core.registry.orthoRequested.template cbits<ORTHO_UNIT, WIDTH>();	}

#if HFSM2_PLANS_AVAILABLE()
	HFSM2_CONSTEXPR(11)	static TaskStatus& headStatus	 (		Control& control )		noexcept	{ return control._core.planData.headStatuses[REGION_ID];	}
	HFSM2_CONSTEXPR(11)	static TaskStatus&  subStatus	 (		Control& control )		noexcept	{ return control._core.planData.subStatuses [REGION_ID];	}
#endif

	HFSM2_CONSTEXPR(14)	void		deepRegister		 (	  Registry& registry, const Parent parent )			noexcept;

	HFSM2_CONSTEXPR(14)	bool		deepForwardEntryGuard(GuardControl& control						  )			noexcept;
	HFSM2_CONSTEXPR(14)	bool		deepEntryGuard		 (GuardControl& control						  )			noexcept;

	HFSM2_CONSTEXPR(14)	void		deepEnter			 ( PlanControl& control						  )			noexcept;
	HFSM2_CONSTEXPR(14)	void		deepReenter			 ( PlanControl& control						  )			noexcept;

	HFSM2_CONSTEXPR(14)	TaskStatus	deepPreUpdate		 ( FullControl& control						  )			noexcept;
	HFSM2_CONSTEXPR(14)	TaskStatus	deepUpdate			 ( FullControl& control						  )			noexcept;
	HFSM2_CONSTEXPR(14)	TaskStatus	deepPostUpdate		 ( FullControl& control						  )			noexcept;

	template <typename TEvent>
	HFSM2_CONSTEXPR(14)	TaskStatus	deepPreReact		 (EventControl& control, const TEvent& event  )			noexcept;

	template <typename TEvent>
	HFSM2_CONSTEXPR(14)	TaskStatus	deepReact			 (EventControl& control, const TEvent& event  )			noexcept;

	template <typename TEvent>
	HFSM2_CONSTEXPR(14)	TaskStatus	deepPostReact		 (EventControl& control, const TEvent& event  )			noexcept;

	template <typename TEvent>
	HFSM2_CONSTEXPR(14)	void		deepQuery			 (ConstControl& control,	   TEvent& event  )	  const noexcept;

#if HFSM2_PLANS_AVAILABLE()
	HFSM2_CONSTEXPR(14)	TaskStatus	deepUpdatePlans		 ( FullControl& control						  )			noexcept;
#endif

	HFSM2_CONSTEXPR(14)	bool		deepForwardExitGuard (GuardControl& control						  )			noexcept;
	HFSM2_CONSTEXPR(14)	bool		deepExitGuard		 (GuardControl& control						  )			noexcept;

	HFSM2_CONSTEXPR(14)	void		deepExit			 ( PlanControl& control						  )			noexcept;

	HFSM2_CONSTEXPR(14)	void		deepForwardActive	 (	   Control& control, const Request request)			noexcept;
	HFSM2_CONSTEXPR(14)	void		deepForwardRequest	 (	   Control& control, const Request request)			noexcept;

	HFSM2_CONSTEXPR(14)	void		deepRequest			 (	   Control& control, const Request request)			noexcept;

	HFSM2_CONSTEXPR(14)	void		deepRequestChange	 (	   Control& control, const Request request)			noexcept;
	HFSM2_CONSTEXPR(14)	void		deepRequestRestart	 (	   Control& control, const Request request)			noexcept;
	HFSM2_CONSTEXPR(14)	void		deepRequestResume	 (	   Control& control, const Request request)			noexcept;
	HFSM2_CONSTEXPR(14)	void		deepRequestSelect	 (	   Control& control, const Request request)			noexcept;

#if HFSM2_UTILITY_THEORY_AVAILABLE()
	HFSM2_CONSTEXPR(14)	void		deepRequestUtilize	 (	   Control& control, const Request request)			noexcept;
	HFSM2_CONSTEXPR(14)	void		deepRequestRandomize (	   Control& control, const Request request)			noexcept;

	HFSM2_CONSTEXPR(14)	UP			deepReportChange	 (	   Control& control						  )			noexcept;

	HFSM2_CONSTEXPR(14)	UP			deepReportUtilize	 (	   Control& control						  )			noexcept;
	HFSM2_CONSTEXPR(14)	Rank		deepReportRank		 (	   Control& control						  )			noexcept;
	HFSM2_CONSTEXPR(14)	Utility		deepReportRandomize  (	   Control& control						  )			noexcept;
#endif

	HFSM2_CONSTEXPR(14)	void		deepChangeToRequested( PlanControl& control						  )			noexcept;

#if HFSM2_SERIALIZATION_AVAILABLE()
	using WriteStream	= typename Args::WriteStream;
	using ReadStream	= typename Args::ReadStream;

	HFSM2_CONSTEXPR(14)	void		deepSaveActive		 (const Registry& registry, WriteStream& stream)  const noexcept;
	HFSM2_CONSTEXPR(14)	void		deepSaveResumable	 (const Registry& registry, WriteStream& stream)  const noexcept;

	HFSM2_CONSTEXPR(14)	void		deepLoadRequested	 (		Registry& registry,  ReadStream& stream)  const noexcept;
	HFSM2_CONSTEXPR(14)	void		deepLoadResumable	 (		Registry& registry,  ReadStream& stream)  const noexcept;
#endif

#if HFSM2_STRUCTURE_REPORT_AVAILABLE()
	using StructureStateInfos = typename Args::StructureStateInfos;

static constexpr Long NAME_COUNT	 = HeadState::NAME_COUNT  + SubStates::NAME_COUNT;

	HFSM2_CONSTEXPR(14)	void deepGetNames(const Long parent,
										  const RegionType region,
										  const Short depth,
										  StructureStateInfos& stateInfos)							  const noexcept;
#endif

};

}
}

namespace hfsm2 {
	namespace detail {

		template <typename TN_, typename TA_, typename TH_, typename... TS_>
		HFSM2_CONSTEXPR(14)
		void
		O_<TN_, TA_, TH_, TS_...>::deepRegister(Registry& registry,
		const Parent parent) noexcept
		{
		registry.orthoParents[ORTHO_INDEX] = parent;
		registry.orthoUnits	 [ORTHO_INDEX] = Units{ORTHO_UNIT, WIDTH};
	registry.regionHeads [REGION_ID]   = HEAD_ID;
	registry.regionSizes [REGION_ID]   = REGION_SIZE;

	HeadState::deepRegister(registry, parent);
	SubStates::wideRegister(registry, ORTHO_ID);
}

template <typename TN_, typename TA_, typename TH_, typename... TS_>
HFSM2_CONSTEXPR(14)
bool
O_<TN_, TA_, TH_, TS_...>::deepForwardEntryGuard(GuardControl& control) noexcept {
const ProngCBits requested = orthoRequested(static_cast<const GuardControl&>(control));

ScopedRegion region{control, REGION_ID, HEAD_ID, REGION_SIZE};

	if (requested)
		return SubStates::wideForwardEntryGuard(control, requested);
	else
		return SubStates::wideForwardEntryGuard(control);
}

template <typename TN_, typename TA_, typename TH_, typename... TS_>
HFSM2_CONSTEXPR(14)
bool
O_<TN_, TA_, TH_, TS_...>::deepEntryGuard(GuardControl& control) noexcept {
ScopedRegion region{control, REGION_ID, HEAD_ID, REGION_SIZE};

	return HeadState::deepEntryGuard(control) ||
		   SubStates::wideEntryGuard(control);
}

template <typename TN_, typename TA_, typename TH_, typename... TS_>
HFSM2_CONSTEXPR(14)
void
O_<TN_, TA_, TH_, TS_...>::deepEnter(PlanControl& control) noexcept {
ProngBits requested = orthoRequested(control);
	requested.clear();

ScopedRegion region{control, REGION_ID, HEAD_ID, REGION_SIZE};

	HeadState::deepEnter(control);
	SubStates::wideEnter(control);
}

template <typename TN_, typename TA_, typename TH_, typename... TS_>
HFSM2_CONSTEXPR(14)
void
O_<TN_, TA_, TH_, TS_...>::deepReenter(PlanControl& control) noexcept {
ProngBits requested = orthoRequested(control);
	requested.clear();

ScopedRegion region{control, REGION_ID, HEAD_ID, REGION_SIZE};

	HeadState::deepReenter(control);
	SubStates::wideReenter(control);
}

template <typename TN_, typename TA_, typename TH_, typename... TS_>
HFSM2_CONSTEXPR(14)
TaskStatus
O_<TN_, TA_, TH_, TS_...>::deepPreUpdate(FullControl& control) noexcept {
ScopedRegion region{control, REGION_ID, HEAD_ID, REGION_SIZE};

const TaskStatus h =
	HeadState::deepPreUpdate(control);
	HFSM2_IF_PLANS(headStatus	(control) |= h);

	HFSM2_IF_PLANS(subStatus	(control) |=)
		SubStates::widePreUpdate(control);

return h;
}

template <typename TN_, typename TA_, typename TH_, typename... TS_>
HFSM2_CONSTEXPR(14)
TaskStatus
O_<TN_, TA_, TH_, TS_...>::deepUpdate(FullControl& control) noexcept {
ScopedRegion region{control, REGION_ID, HEAD_ID, REGION_SIZE};

const TaskStatus h =
	HeadState::deepUpdate(control);
	HFSM2_IF_PLANS(headStatus(control) |= h);

	HFSM2_IF_PLANS(subStatus (control) |=)
		SubStates::wideUpdate(control);

return h;
}

template <typename TN_, typename TA_, typename TH_, typename... TS_>
HFSM2_CONSTEXPR(14)
TaskStatus
O_<TN_, TA_, TH_, TS_...>::deepPostUpdate(FullControl& control) noexcept {
ScopedRegion region{control, REGION_ID, HEAD_ID, REGION_SIZE};

	HFSM2_IF_PLANS(subStatus	 (control) |=)
		SubStates::widePostUpdate(control);

const TaskStatus h =
	HeadState::deepPostUpdate(control);
	HFSM2_IF_PLANS(headStatus	 (control) |= h);

return h;
}

template <typename TN_, typename TA_, typename TH_, typename... TS_>
template <typename TEvent>
HFSM2_CONSTEXPR(14)
TaskStatus
O_<TN_, TA_, TH_, TS_...>::deepPreReact(EventControl& control,
										const TEvent& event) noexcept
{
ScopedRegion region{control, REGION_ID, HEAD_ID, REGION_SIZE};

	return PreReactWrapper::execute(*this, control, event);
}

template <typename TN_, typename TA_, typename TH_, typename... TS_>
template <typename TEvent>
HFSM2_CONSTEXPR(14)
TaskStatus
O_<TN_, TA_, TH_, TS_...>::deepReact(EventControl& control,
									 const TEvent& event) noexcept
{
ScopedRegion region{control, REGION_ID, HEAD_ID, REGION_SIZE};

	return ReactWrapper::execute(*this, control, event);
}

template <typename TN_, typename TA_, typename TH_, typename... TS_>
template <typename TEvent>
HFSM2_CONSTEXPR(14)
TaskStatus
O_<TN_, TA_, TH_, TS_...>::deepPostReact(EventControl& control,
										 const TEvent& event) noexcept
{
ScopedRegion region{control, REGION_ID, HEAD_ID, REGION_SIZE};

	return PostReactWrapper::execute(*this, control, event);
}

template <typename TN_, typename TA_, typename TH_, typename... TS_>
template <typename TEvent>
HFSM2_CONSTEXPR(14)
void
O_<TN_, TA_, TH_, TS_...>::deepQuery(ConstControl& control,
									 TEvent& event) const noexcept
{
ScopedCRegion region{control, REGION_ID};

	QueryWrapper::execute(*this, control, event);
}

#if HFSM2_PLANS_AVAILABLE()

template <typename TN_, typename TA_, typename TH_, typename... TS_>
HFSM2_CONSTEXPR(14)
TaskStatus
O_<TN_, TA_, TH_, TS_...>::deepUpdatePlans(FullControl& control) noexcept {
	const TaskStatus h = headStatus(control) |
		HeadState::deepUpdatePlans (control);

	const TaskStatus s =  subStatus(control) |
		SubStates::wideUpdatePlans (control);

	if (h)
		return h;
	else {
		if (s.outerTransition)
			return TaskStatus{TaskStatus::NONE, true};

		ScopedRegion region{control, REGION_ID, HEAD_ID, REGION_SIZE};

		const bool planExists = control._core.planData.planExists.template get<REGION_ID>();

		return s && planExists ?
			control.updatePlan(static_cast<HeadState&>(*this), s) : s;
	}
}

#endif

template <typename TN_, typename TA_, typename TH_, typename... TS_>
HFSM2_CONSTEXPR(14)
bool
O_<TN_, TA_, TH_, TS_...>::deepForwardExitGuard(GuardControl& control) noexcept {
const ProngCBits requested = orthoRequested(static_cast<const GuardControl&>(control));

ScopedRegion region{control, REGION_ID, HEAD_ID, REGION_SIZE};

	if (requested)
		return SubStates::wideForwardExitGuard(control, requested);
	else
		return SubStates::wideForwardExitGuard(control);
}

template <typename TN_, typename TA_, typename TH_, typename... TS_>
HFSM2_CONSTEXPR(14)
bool
O_<TN_, TA_, TH_, TS_...>::deepExitGuard(GuardControl& control) noexcept {
ScopedRegion region{control, REGION_ID, HEAD_ID, REGION_SIZE};

	return SubStates::wideExitGuard(control) ||
		   HeadState::deepExitGuard(control);
}

template <typename TN_, typename TA_, typename TH_, typename... TS_>
HFSM2_CONSTEXPR(14)
void
O_<TN_, TA_, TH_, TS_...>::deepExit(PlanControl& control) noexcept {
	SubStates::wideExit(control);
	HeadState::deepExit(control);
}

template <typename TN_, typename TA_, typename TH_, typename... TS_>
HFSM2_CONSTEXPR(14)
void
O_<TN_, TA_, TH_, TS_...>::deepForwardActive(Control& control,
											 const Request request) noexcept
{
	HFSM2_ASSERT(control._core.registry.isActive(HEAD_ID));

const ProngCBits requested = orthoRequested(static_cast<const Control&>(control));
	HFSM2_ASSERT(!!requested);

	SubStates::wideForwardActive(control, request, requested);
}

template <typename TN_, typename TA_, typename TH_, typename... TS_>
HFSM2_CONSTEXPR(14)
void
O_<TN_, TA_, TH_, TS_...>::deepForwardRequest(Control& control,
											  const Request request) noexcept
{
	HFSM2_IF_TRANSITION_HISTORY(control.pinLastTransition(HEAD_ID, request.index));

const ProngCBits requested = orthoRequested(static_cast<const Control&>(control));

	if (requested)
		SubStates::wideForwardRequest(control, request);
	else
		deepRequest					 (control, request);
}

template <typename TN_, typename TA_, typename TH_, typename... TS_>
HFSM2_CONSTEXPR(14)
void
O_<TN_, TA_, TH_, TS_...>::deepRequest(Control& control,
									   const Request request) noexcept
{
	switch (request.type) {
	case TransitionType::CHANGE:
		deepRequestChange	(control, request);
		break;

	case TransitionType::RESTART:
		deepRequestRestart	(control, request);
		break;

	case TransitionType::RESUME:
		deepRequestResume	(control, request);
		break;

	case TransitionType::SELECT:
		deepRequestSelect	(control, request);
		break;

#if HFSM2_UTILITY_THEORY_AVAILABLE()

	case TransitionType::UTILIZE:
		deepRequestUtilize	(control, request);
		break;

	case TransitionType::RANDOMIZE:
		deepRequestRandomize(control, request);
		break;

#endif

	default:
		HFSM2_BREAK();
	}
}

template <typename TN_, typename TA_, typename TH_, typename... TS_>
HFSM2_CONSTEXPR(14)
void
O_<TN_, TA_, TH_, TS_...>::deepRequestChange(Control& control,
											 const Request request) noexcept
{
	HFSM2_IF_TRANSITION_HISTORY(control.pinLastTransition(HEAD_ID, request.index));

	SubStates::wideRequestChange(control, request);
}

template <typename TN_, typename TA_, typename TH_, typename... TS_>
HFSM2_CONSTEXPR(14)
void
O_<TN_, TA_, TH_, TS_...>::deepRequestRestart(Control& control,
											  const Request request) noexcept
{
	HFSM2_IF_TRANSITION_HISTORY(control.pinLastTransition(HEAD_ID, request.index));

	SubStates::wideRequestRestart(control, request);
}

template <typename TN_, typename TA_, typename TH_, typename... TS_>
HFSM2_CONSTEXPR(14)
void
O_<TN_, TA_, TH_, TS_...>::deepRequestResume(Control& control,
											 const Request request) noexcept
{
	HFSM2_IF_TRANSITION_HISTORY(control.pinLastTransition(HEAD_ID, request.index));

	SubStates::wideRequestResume(control, request);
}

template <typename TN_, typename TA_, typename TH_, typename... TS_>
HFSM2_CONSTEXPR(14)
void
O_<TN_, TA_, TH_, TS_...>::deepRequestSelect(Control& control,
											 const Request request) noexcept
{
	HFSM2_IF_TRANSITION_HISTORY(control.pinLastTransition(HEAD_ID, request.index));

	SubStates::wideRequestSelect(control, request);
}

#if HFSM2_UTILITY_THEORY_AVAILABLE()

template <typename TN_, typename TA_, typename TH_, typename... TS_>
HFSM2_CONSTEXPR(14)
void
O_<TN_, TA_, TH_, TS_...>::deepRequestUtilize(Control& control,
											  const Request request) noexcept
{
	HFSM2_IF_TRANSITION_HISTORY(control.pinLastTransition(HEAD_ID, request.index));

	SubStates::wideRequestUtilize(control, request);
}

template <typename TN_, typename TA_, typename TH_, typename... TS_>
HFSM2_CONSTEXPR(14)
void
O_<TN_, TA_, TH_, TS_...>::deepRequestRandomize(Control& control,
												const Request request) noexcept
{
	HFSM2_IF_TRANSITION_HISTORY(control.pinLastTransition(HEAD_ID, request.index));

	SubStates::wideRequestRandomize(control, request);
}

template <typename TN_, typename TA_, typename TH_, typename... TS_>
HFSM2_CONSTEXPR(14)
typename TA_::UP
O_<TN_, TA_, TH_, TS_...>::deepReportChange(Control& control) noexcept {
const UP	  h = HeadState::deepReportChange(control);
const Utility s = SubStates::wideReportChange(control);

const Utility sub = s / WIDTH;

	HFSM2_LOG_UTILITY_RESOLUTION(control.context(), HEAD_ID, INVALID_SHORT, sub);

	return {
h.utility * sub,
		h.prong
	};
}

template <typename TN_, typename TA_, typename TH_, typename... TS_>
HFSM2_CONSTEXPR(14)
typename TA_::UP
O_<TN_, TA_, TH_, TS_...>::deepReportUtilize(Control& control) noexcept {
const UP	  h = HeadState::deepReportUtilize(control);
const Utility s = SubStates::wideReportUtilize(control);

const Utility sub = s / WIDTH;

	HFSM2_LOG_UTILITY_RESOLUTION(control.context(), HEAD_ID, INVALID_SHORT, sub);

	return {
h.utility * sub,
		h.prong
	};
}

template <typename TN_, typename TA_, typename TH_, typename... TS_>
HFSM2_CONSTEXPR(14)
typename TA_::Rank
O_<TN_, TA_, TH_, TS_...>::deepReportRank(Control& control) noexcept {
	return HeadState::wrapRank(control);
}

template <typename TN_, typename TA_, typename TH_, typename... TS_>
HFSM2_CONSTEXPR(14)
typename TA_::Utility
O_<TN_, TA_, TH_, TS_...>::deepReportRandomize(Control& control) noexcept {
const Utility h = HeadState::wrapUtility(control);
const Utility s = SubStates::wideReportRandomize(control);

const Utility sub = s / WIDTH;

	HFSM2_LOG_RANDOM_RESOLUTION(control.context(), HEAD_ID, INVALID_SHORT, sub);

return h * sub;
}

#endif

template <typename TN_, typename TA_, typename TH_, typename... TS_>
HFSM2_CONSTEXPR(14)
void
O_<TN_, TA_, TH_, TS_...>::deepChangeToRequested(PlanControl& control) noexcept {
	SubStates::wideChangeToRequested(control);
}

#if HFSM2_SERIALIZATION_AVAILABLE()

template <typename TN_, typename TA_, typename TH_, typename... TS_>
HFSM2_CONSTEXPR(14)
void
O_<TN_, TA_, TH_, TS_...>::deepSaveActive(const Registry& registry,
										  WriteStream& stream) const noexcept
{
	SubStates::wideSaveActive(registry, stream);
}

template <typename TN_, typename TA_, typename TH_, typename... TS_>
HFSM2_CONSTEXPR(14)
void
O_<TN_, TA_, TH_, TS_...>::deepSaveResumable(const Registry& registry,
											 WriteStream& stream) const noexcept
{
	SubStates::wideSaveResumable(registry, stream);
}

template <typename TN_, typename TA_, typename TH_, typename... TS_>
HFSM2_CONSTEXPR(14)
void
O_<TN_, TA_, TH_, TS_...>::deepLoadRequested(Registry& registry,
											 ReadStream& stream) const noexcept
{
	SubStates::wideLoadRequested(registry, stream);
}

template <typename TN_, typename TA_, typename TH_, typename... TS_>
HFSM2_CONSTEXPR(14)
void
O_<TN_, TA_, TH_, TS_...>::deepLoadResumable(Registry& registry,
											 ReadStream& stream) const noexcept
{
	SubStates::wideLoadResumable(registry, stream);
}

#endif

#if HFSM2_STRUCTURE_REPORT_AVAILABLE()

template <typename TN_, typename TA_, typename TH_, typename... TS_>
HFSM2_CONSTEXPR(14)
void
O_<TN_, TA_, TH_, TS_...>::deepGetNames(const Long parent,
										const RegionType region,
										const Short depth,
										StructureStateInfos& stateInfos) const noexcept
{
	HeadState::deepGetNames(parent, region,			depth,	   stateInfos);
	SubStates::wideGetNames(stateInfos.count() - 1, depth + 1, stateInfos);
}

#endif

}
}

namespace hfsm2 {
	namespace detail {

		template <
		FeatureTag NFeatureTag
		, typename TContext
		, typename TActivation
		, typename TReactOrder

#if HFSM2_UTILITY_THEORY_AVAILABLE()
		, typename TRank
		, typename TUtility
		, typename TRNG
#endif

		, Short NSubstitutionLimit
		HFSM2_IF_PLANS(, Long NTaskCapacity)
		, typename TPayload
		>
		struct G_ final {
		static constexpr FeatureTag FEATURE_TAG = NFeatureTag;

		using Context			 = TContext;
		using Activation		 = TActivation;
		using ReactOrder		 = TReactOrder;

#if HFSM2_UTILITY_THEORY_AVAILABLE()
		using Rank				 = TRank;
		using Utility			 = TUtility;
		using RNG				 = TRNG;
#endif

		static constexpr Short SUBSTITUTION_LIMIT = NSubstitutionLimit;

#if HFSM2_PLANS_AVAILABLE()
		static constexpr Long TASK_CAPACITY		  = NTaskCapacity;
#endif

		using Payload			 = TPayload;
		using Transition		 = TransitionT<Payload>;

#if HFSM2_PLANS_AVAILABLE()
		using Task				 = TaskT<Payload>;
#endif

#if HFSM2_LOG_INTERFACE_AVAILABLE()
		using LoggerInterface	 = LoggerInterfaceT<FEATURE_TAG, Context HFSM2_IF_UTILITY_THEORY(, Utility)>;
#endif

		/// @brief Set Context type
		/// @tparam `T` Context type for data shared between states and/or data interface between FSM and external code
		template <typename T>
		using ContextT			 = G_<FEATURE_TAG, T	  , Activation, ReactOrder HFSM2_IF_UTILITY_THEORY(, Rank, Utility, RNG), SUBSTITUTION_LIMIT HFSM2_IF_PLANS(, TASK_CAPACITY), Payload>;

		/// @brief Select manual activation strategy
		using ManualActivation	 = G_<FEATURE_TAG, Context, Manual	  , ReactOrder HFSM2_IF_UTILITY_THEORY(, Rank, Utility, RNG), SUBSTITUTION_LIMIT HFSM2_IF_PLANS(, TASK_CAPACITY), Payload>;

		/// @brief Select event processing order
		using BottomUpReactions	 = G_<FEATURE_TAG, Context, Activation, BottomUp   HFSM2_IF_UTILITY_THEORY(, Rank, Utility, RNG), SUBSTITUTION_LIMIT HFSM2_IF_PLANS(, TASK_CAPACITY), Payload>;

#if HFSM2_UTILITY_THEORY_AVAILABLE()

		/// @brief Set Rank type
		/// @tparam `T` Rank type for 'TRank State::rank() const' method
		template <typename T>
		using RankT				 = G_<FEATURE_TAG, Context, Activation, ReactOrder						   , T   , Utility, RNG , SUBSTITUTION_LIMIT HFSM2_IF_PLANS(, TASK_CAPACITY), Payload>;

		/// @brief Set Utility type
		/// @tparam `T` Utility type for 'TUtility State::utility() const' method
		template <typename T>
		using UtilityT			 = G_<FEATURE_TAG, Context, Activation, ReactOrder						   , Rank, T      , RNG , SUBSTITUTION_LIMIT HFSM2_IF_PLANS(, TASK_CAPACITY), Payload>;

		/// @brief Set RNG type
		/// @tparam `T` RNG type used in 'Random' regions
		template <typename T>
		using RandomT			 = G_<FEATURE_TAG, Context, Activation, ReactOrder						   , Rank, Utility, T   , SUBSTITUTION_LIMIT HFSM2_IF_PLANS(, TASK_CAPACITY), Payload>;

#endif

		/// @brief Set Substitution limit
		/// @tparam `N` Maximum number times 'guard()' methods can substitute their states for others
		template <Short N>
		using SubstitutionLimitN = G_<FEATURE_TAG, Context, Activation, ReactOrder HFSM2_IF_UTILITY_THEORY(, Rank, Utility, RNG), N                  HFSM2_IF_PLANS(, TASK_CAPACITY), Payload>;

#if HFSM2_PLANS_AVAILABLE()

		/// @brief Set Task capacity
		/// @tparam `N` Maximum number of tasks across all plans
		template <Long N>
		using TaskCapacityN		 = G_<FEATURE_TAG, Context, Activation, ReactOrder HFSM2_IF_UTILITY_THEORY(, Rank, Utility, RNG), SUBSTITUTION_LIMIT                , N             , Payload>;

#endif

		/// @brief Set Transition Payload type
		/// @tparam `T` Payload type
		template <typename T>
		using PayloadT			 = G_<FEATURE_TAG, Context, Activation, ReactOrder HFSM2_IF_UTILITY_THEORY(, Rank, Utility, RNG), SUBSTITUTION_LIMIT HFSM2_IF_PLANS(, TASK_CAPACITY), T      >;

#if HFSM2_UTILITY_THEORY_AVAILABLE()

		struct UP final {
		HFSM2_CONSTEXPR(14)	UP(const Utility utility_ = Utility{1},
		const Prong prong_ = INVALID_PRONG)		noexcept
	: utility{utility_}
, prong{prong_}
		{}

Utility utility;
Prong prong;
	};

#endif

};

template <typename>
struct M_;

template <
	FeatureTag NFeatureTag
  , typename TContext
  , typename TActivation
  , typename TReactOrder

#if HFSM2_UTILITY_THEORY_AVAILABLE()
, typename TRank
, typename TUtility
  , typename TRNG
#endif

, Short NSubstitutionLimit
  HFSM2_IF_PLANS(, Long NTaskCapacity)
  , typename TPayload
>
struct M_<
		   G_<
			   NFeatureTag
			 , TContext
			 , TActivation
			 , TReactOrder
			 HFSM2_IF_UTILITY_THEORY(, TRank, TUtility, TRNG)
			 , NSubstitutionLimit
			 HFSM2_IF_PLANS(, NTaskCapacity)
			 , TPayload
		   >
	   > final
{
	using Cfg = G_<
	NFeatureTag
	, TContext
	, TActivation
	, TReactOrder
				  HFSM2_IF_UTILITY_THEORY(, TRank, TUtility, TRNG)
				  , NSubstitutionLimit
				  HFSM2_IF_PLANS(, NTaskCapacity)
				  , TPayload
				>;

static constexpr FeatureTag FEATURE_TAG = NFeatureTag;

	using Context			= TContext;

#if HFSM2_UTILITY_THEORY_AVAILABLE()
	using Utility			= TUtility;
#endif

	using Payload			= TPayload;
using Transition		= TransitionT<Payload>;

#if HFSM2_LOG_INTERFACE_AVAILABLE()
	using LoggerInterface	= typename Cfg::LoggerInterface;
#endif

	/// @brief Composite region ('changeTo<>()' into the region acts as 'restart<>()')
	/// @tparam THead Head state
	/// @tparam TSubStates Sub-states
	template <typename THead, typename... TSubStates>
	using Composite			 = CI_<Strategy::Composite,	   THead, TSubStates...>;

	/// @brief Headless composite region ('changeTo<>()' into the region acts as 'restart<>()')
	/// @tparam TSubStates Sub-states
	template <				  typename... TSubStates>
	using CompositePeers	 = CI_<Strategy::Composite,    void,  TSubStates...>;

	/// @brief Resumable region ('changeTo<>()' into the region acts as 'resume<>()')
	/// @tparam THead Head state
	/// @tparam TSubStates Sub-states
	template <typename THead, typename... TSubStates>
	using Resumable			  = CI_<Strategy::Resumable,   THead, TSubStates...>;

	/// @brief Headless resumable region ('changeTo<>()' into the region acts as 'resume<>()')
	/// @tparam TSubStates Sub-states
	template <				  typename... TSubStates>
	using ResumablePeers	  = CI_<Strategy::Resumable,   void,  TSubStates...>;

	/// @brief Selectable region ('changeTo<>()' into the region acts as 'select<>()')
	/// @tparam THead Head state
	/// @tparam TSubStates Sub-states
	template <typename THead, typename... TSubStates>
	using Selectable		  = CI_<Strategy::Selectable,  THead, TSubStates...>;

	/// @brief Headless selectable region ('changeTo<>()' into the region acts as 'select<>()')
	/// @tparam TSubStates Sub-states
	template <				  typename... TSubStates>
	using SelectablePeers	  = CI_<Strategy::Selectable,  void,  TSubStates...>;

#if HFSM2_UTILITY_THEORY_AVAILABLE()

	/// @brief Utilitarian region ('changeTo<>()' into the region acts as 'utilize<>()')
	/// @tparam THead Head state
	/// @tparam TSubStates Sub-states
	template <typename THead, typename... TSubStates>
	using Utilitarian		  = CI_<Strategy::Utilitarian, THead, TSubStates...>;

	/// @brief Headless utilitarian region ('changeTo<>()' into the region acts as 'utilize<>()')
	/// @tparam TSubStates Sub-states
	template <				  typename... TSubStates>
	using UtilitarianPeers	  = CI_<Strategy::Utilitarian, void,  TSubStates...>;

	/// @brief Random region ('changeTo<>()' into the region acts as 'randomize<>()')
	/// @tparam THead Head state
	/// @tparam TSubStates Sub-states
	template <typename THead, typename... TSubStates>
	using Random			  = CI_<Strategy::RandomUtil,  THead, TSubStates...>;

	/// @brief Headless random region ('changeTo<>()' into the region acts as 'randomize<>()')
	/// @tparam TSubStates Sub-states
	template <				  typename... TSubStates>
	using RandomPeers		  = CI_<Strategy::RandomUtil,  void,  TSubStates...>;

#endif

	/// @brief Orthogonal region (when activated, activates all sub-states)
	/// @tparam THead Head state
	/// @tparam TSubStates Sub-states
	template <typename THead, typename... TSubStates>
	using Orthogonal		  = OI_<THead, TSubStates...>;

	/// @brief Headless orthogonal region (when activated, activates all sub-states)
	/// @tparam TSubStates Sub-states
	template <				  typename... TSubStates>
	using OrthogonalPeers	  = OI_<void,  TSubStates...>;

	/// @brief Root ('changeTo<>()' into the root region acts as 'restart<>()')
	/// @tparam THead Head state
	/// @tparam TSubStates Sub-states
	template <typename THead, typename... TSubStates>
	using Root				  = RF_<Cfg, Composite  <THead, TSubStates...>>;

	/// @brief Headless root ('changeTo<>()' into the root region acts as 'restart<>()')
	/// @tparam TSubStates Sub-states
	template <				  typename... TSubStates>
	using PeerRoot			  = RF_<Cfg, CompositePeers  <  TSubStates...>>;

	/// @brief Resumable root ('changeTo<>()' into the root region acts as 'resume<>()')
	/// @tparam THead Head state
	/// @tparam TSubStates Sub-states
	template <typename THead, typename... TSubStates>
	using ResumableRoot		  = RF_<Cfg, Resumable  <THead, TSubStates...>>;

	/// @brief Headless resumable root ('changeTo<>()' into the root region acts as 'resume<>()')
	/// @tparam TSubStates Sub-states
	template <				  typename... TSubStates>
	using ResumablePeerRoot	  = RF_<Cfg, ResumablePeers  <  TSubStates...>>;

	/// @brief Selectable root ('changeTo<>()' into the region acts as 'select<>()')
	/// @tparam THead Head state
	/// @tparam TSubStates Sub-states
	template <typename THead, typename... TSubStates>
	using SelectableRoot	  = RF_<Cfg, Selectable <THead, TSubStates...>>;

	/// @brief Headless selectable root ('changeTo<>()' into the region acts as 'select<>()')
	/// @tparam TSubStates Sub-states
	template <				  typename... TSubStates>
	using SelectablePeerRoot  = RF_<Cfg, SelectablePeers <  TSubStates...>>;

#if HFSM2_UTILITY_THEORY_AVAILABLE()

	/// @brief Utilitarian root ('changeTo<>()' into the root region acts as 'utilize<>()')
	/// @tparam THead Head state
	/// @tparam TSubStates Sub-states
	template <typename THead, typename... TSubStates>
	using UtilitarianRoot	  = RF_<Cfg, Utilitarian<THead, TSubStates...>>;

	/// @brief Headless utilitarian root ('changeTo<>()' into the root region acts as 'utilize<>()')
	/// @tparam TSubStates Sub-states
	template <				  typename... TSubStates>
	using UtilitarianPeerRoot = RF_<Cfg, UtilitarianPeers<  TSubStates...>>;

	/// @brief Random root ('changeTo<>()' into the root region acts as 'randomize<>()')
	/// @tparam THead Head state
	/// @tparam TSubStates Sub-states
	template <typename THead, typename... TSubStates>
	using RandomRoot		  = RF_<Cfg, Random		<THead, TSubStates...>>;

	/// @brief Headless random root ('changeTo<>()' into the root region acts as 'randomize<>()')
	/// @tparam TSubStates Sub-states
	template <				  typename... TSubStates>
	using RandomPeerRoot	  = RF_<Cfg, RandomPeers	 <  TSubStates...>>;

#endif

	/// @brief Orthogonal root (all sub-states are active at all times)
	/// @tparam THead Head state
	/// @tparam TSubStates Sub-states
	template <typename THead, typename... TSubStates>
	using OrthogonalRoot	  = RF_<Cfg, Orthogonal <THead, TSubStates...>>;

	/// @brief Headless orthogonal root (all sub-states are active at all times)
	/// @tparam TSubStates Sub-states
	template <				  typename... TSubStates>
	using OrthogonalPeerRoot  = RF_<Cfg, OrthogonalPeers <  TSubStates...>>;

};

}

/// @brief Type configuration for MachineT<>
using Config = detail::G_<
	HFSM2_FEATURE_TAG
	, EmptyContext
	, Automatic
	, TopDown
						 HFSM2_IF_UTILITY_THEORY(, int8_t, float, RNGT<float>)
						 , 4
						 HFSM2_IF_PLANS(, INVALID_LONG)
						 , void
					   >;

/// @brief 'Template namespace' for FSM classes
/// @tparam `TConfig` `ConfigT<>` type configuration for MachineT<>
/// @see `ConfigT<>`
template <typename TConfig = Config>
using MachineT = detail::M_<TConfig>;

/// @brief 'Template namespace' for FSM classes parametrized with default types
using Machine = MachineT<>;

}

namespace hfsm2 {
	namespace detail {

		/// @brief FSM Root
		/// @tparam Cfg Type configuration
		/// @tparam TApex Root region type
		template <
		typename TConfig
		, typename TApex
		>
		class R_ {
			public:
			static constexpr FeatureTag FEATURE_TAG = TConfig::FEATURE_TAG;

			using Context				= typename TConfig::Context;

#if HFSM2_UTILITY_THEORY_AVAILABLE()
			using Rank					= typename TConfig::Rank;
			using Utility				= typename TConfig::Utility;
			using RNG					= typename TConfig::RNG;
#endif

			using Payload				= typename TConfig::Payload;

			protected:
			using Forward				= RF_<TConfig, TApex>;
			using StateList				= typename Forward::StateList;
			using RegionList			= typename Forward::RegionList;

			static constexpr Long STATE_COUNT	= StateList ::SIZE;
			static constexpr Long REGION_COUNT	= RegionList::SIZE;

			using Args					= typename Forward::Args;
			using PureContext			= typename Args::PureContext;

			static_assert(Args::STATE_COUNT	   < static_cast<unsigned>(-1), "Too many states in the FSM. Change 'Short' type.");
			static_assert(Args::STATE_COUNT	  == static_cast<unsigned>(StateList::SIZE), "STATE_COUNT != StateList::SIZE");
			static_assert(Args::COMPO_COUNT >= 1, "State machine needs at least one composite region");

			using Core					= CoreT<Args>;

			using Apex					= MaterialT<I_<0, 0, 0, 0>, Args, TApex>;

			using Registry				= RegistryT<Args>;
			using CompoForks			= typename Registry::CompoForks;
			using RegistryBackUp		= typename Registry::BackUp;

			using ConstControl			= ConstControlT<Args>;
			using Control				= ControlT	   <Args>;
			using PlanControl			= PlanControlT <Args>;
			using FullControl			= FullControlT <Args>;
			using GuardControl			= GuardControlT<Args>;
			using EventControl			= EventControlT<Args>;

			static constexpr Short	SUBSTITUTION_LIMIT	= Forward::SUBSTITUTION_LIMIT;

#if HFSM2_PLANS_AVAILABLE()
			using PlanData				= PlanDataT<Args>;
#endif

			public:
#if HFSM2_SERIALIZATION_AVAILABLE()
			using WriteStream			= typename Args::WriteStream;
			using ReadStream			= typename Args::ReadStream;
#endif

#if HFSM2_STRUCTURE_REPORT_AVAILABLE()
			static constexpr Long NAME_COUNT = Apex::NAME_COUNT;
#endif

			public:
			using Info					= WrapInfo<TApex>;

			/// @brief Transition
			using Transition			= typename Core::Transition;

			/// @brief Array of transitions
			using TransitionSet			= typename Control::TransitionSet;
			using TransitionSets		= typename Control::TransitionSets;

#if HFSM2_PLANS_AVAILABLE()
			using CPlan					= CPlanT<Args>;
			using Plan					= PayloadPlanT<Args>;

			static constexpr Long TASK_CAPACITY = Forward::TASK_CAPACITY;
#endif

#if HFSM2_TRANSITION_HISTORY_AVAILABLE()
			using TransitionTargets		= typename Control::TransitionTargets;
#endif

#if HFSM2_STRUCTURE_REPORT_AVAILABLE()
			using Prefix				= StaticArrayT<wchar_t, Info::REVERSE_DEPTH * 2 + 2>;
			using Prefixes				= StaticArrayT<Prefix, STATE_COUNT>;

			using NamedStates			= BitArrayT<STATE_COUNT>;

			using StructureStateInfos	= typename Args::StructureStateInfos;
#endif

#if HFSM2_LOG_INTERFACE_AVAILABLE()
			using Logger				= typename TConfig::LoggerInterface;
#endif

			public:

			HFSM2_CONSTEXPR(14)	explicit R_(Context& context
			HFSM2_IF_UTILITY_THEORY(, RNG& rng)
			HFSM2_IF_LOG_INTERFACE(, Logger* const logger = nullptr))		noexcept;

			HFSM2_CONSTEXPR(14)	explicit R_(PureContext&& context
			HFSM2_IF_UTILITY_THEORY(, RNG& rng)
			HFSM2_IF_LOG_INTERFACE(, Logger* const logger = nullptr))		noexcept;

			HFSM2_CONSTEXPR(NO) R_(const R_& )															noexcept = default;
			HFSM2_CONSTEXPR(NO) R_(		 R_&&)															noexcept = default;

			HFSM2_CONSTEXPR(20)	~R_()																	noexcept;

			/// @brief Get state identifier for a state type
			/// @tparam `TState` State type
			/// @return Numeric state identifier
			template <typename TState>
			static
		HFSM2_CONSTEXPR(11) StateID  stateId()														noexcept	{ return					   index<StateList , TState>() ;	}

		/// @brief Get region identifier for a region type
		/// @tparam `TState` Region head state type
		/// @return Numeric region identifier
		template <typename TState>
		static
	HFSM2_CONSTEXPR(11) RegionID regionId()														noexcept	{ return static_cast<RegionID>(index<RegionList, TState>());	}

	/// @brief Access context
	/// @return context
HFSM2_CONSTEXPR(14)		  Context& context()												noexcept	{ return _core.context;							}

	/// @brief Access context
	/// @return context
	HFSM2_CONSTEXPR(11)	const Context& context()										  const noexcept	{ return _core.context;							}

	/// @brief Access state instance
	/// @tparam `TState` State type
	/// @return State instance
	template <typename TState>
	HFSM2_CONSTEXPR(14)		  TState& access()													noexcept	{ return static_cast<	   TState&>(_apex);		}

	/// @brief Access state instance
	/// @tparam `TState` State type
	/// @return State instance
	template <typename TState>
	HFSM2_CONSTEXPR(11)	const TState& access()											  const noexcept	{ return static_cast<const TState&>(_apex);		}

	/// @brief Trigger FSM update cycle (recursively call `update()` from the root down to the leaf states
	///   on all active states then process requested transitions)
	HFSM2_CONSTEXPR(14)	void update()															noexcept;

	/// @brief Have FSM react to an event (recursively call matching 'react<>()' from the root down to the leaf states
	///   on all active states then process requested transitions)
	/// @tparam `TEvent` Event type
	/// @param `event` Event to react to
	template <typename TEvent>
	HFSM2_CONSTEXPR(14)	void react(const TEvent& event)											noexcept;

	/// @brief Recursively call 'query()' from the root down to the leaf states on all active states
	/// @tparam `TEvent` Event type
	/// @param `event` Event to react to
	template <typename TEvent>
	HFSM2_CONSTEXPR(14)	void query(TEvent& event)										  const noexcept;

	/// @brief Get region's active sub-state's index
	/// @param `stateId` Region's head state identifier
	/// @return Region's active sub-state index
	HFSM2_CONSTEXPR(14)	Prong activeSubState (const StateID stateId_)					  const noexcept	{ return _core.registry.activeSubState(stateId_			);	}

	/// @brief Get region's active sub-state's index
	/// @tparam `TState` Region's head state type
	/// @return Region's active sub-state index
	template <typename TState>
	HFSM2_CONSTEXPR(14)	Prong activeSubState ()											  const noexcept	{ return _core.registry.activeSubState(stateId<TState>());	}

	/// @brief Check if a state is active
	/// @param `stateId` Destination state identifier
	/// @return State active status
	HFSM2_CONSTEXPR(11)	bool isActive		 (const StateID stateId_)					  const noexcept	{ return _core.registry.isActive   (stateId_);				}

	/// @brief Check if a state is active
	/// @tparam `TState` Destination state type
	/// @return State active status
	template <typename TState>
	HFSM2_CONSTEXPR(11)	bool isActive		 ()											  const noexcept	{ return isActive	(stateId<TState>());					}

	/// @brief Check if a state is resumable (activated then deactivated previously)
	/// @param `stateId` Destination state identifier
	/// @return State resumable status
	HFSM2_CONSTEXPR(11)	bool isResumable	 (const StateID stateId_)					  const noexcept	{ return _core.registry.isResumable(stateId_);				}

	/// @brief Check if a state is resumable (activated then deactivated previously)
	/// @tparam `TState` Destination state type
	/// @return State resumable status
	template <typename TState>
	HFSM2_CONSTEXPR(11)	bool isResumable	 ()											  const noexcept	{ return isResumable(stateId<TState>());					}

	/// @brief Check if a state is scheduled to activate on the next transition to parent region
	/// @param `stateId` Destination state identifier
	/// @return State scheduled status
	HFSM2_CONSTEXPR(11)	bool isScheduled	 (const StateID stateId_)					  const noexcept	{ return isResumable(stateId_);								}

	/// @brief Check if a state is scheduled to activate on the next transition to parent region
	/// @tparam `TState` Destination state type
	/// @return State scheduled status
	template <typename TState>
	HFSM2_CONSTEXPR(11)	bool isScheduled	 ()											  const noexcept	{ return isResumable<TState>();								}

#if HFSM2_PLANS_AVAILABLE()

	/// @brief Access plan for the root region
	/// @return Plan for the root region
	/// @see `HFSM2_ENABLE_PLANS`
	HFSM2_CONSTEXPR(14)  Plan plan()															noexcept	{ return  Plan{_core.registry, _core.planData, 0				  };	}

	/// @brief Access plan for a region
	/// @param `regionId` Region identifier
	/// @return Plan for the region
	/// @see `HFSM2_ENABLE_PLANS`
	HFSM2_CONSTEXPR(14)  Plan plan(const RegionID regionId_)									noexcept	{ return  Plan{_core.registry, _core.planData, regionId_		  };	}

	/// @brief Access plan for a region
	/// @tparam `TRegion` Region head state type
	/// @return Plan for the region
	/// @see `HFSM2_ENABLE_PLANS`
	template <typename TRegion>
	HFSM2_CONSTEXPR(14)  Plan plan()															noexcept	{ return  Plan{_core.registry, _core.planData, regionId<TRegion>()};	}

	/// @brief Access read-only plan for the root region
	/// @return Read-only plan for the root region
	/// @see `HFSM2_ENABLE_PLANS`
	HFSM2_CONSTEXPR(11)	CPlan plan()													  const noexcept	{ return CPlan{_core.registry, _core.planData, 0				  };	}

	/// @brief Access read-only plan for a region
	/// @param `regionId` Region identifier
	/// @return Read-only plan for the region
	/// @see `HFSM2_ENABLE_PLANS`
	HFSM2_CONSTEXPR(11)	CPlan plan(const RegionID regionId_)							  const noexcept	{ return CPlan{_core.registry, _core.planData, regionId_		  };	}

	/// @brief Access plan for a region
	/// @tparam `TRegion` Region head state type
	/// @return Plan for the region
	/// @see `HFSM2_ENABLE_PLANS`
	template <typename TRegion>
	HFSM2_CONSTEXPR(11)	CPlan plan()													  const noexcept	{ return CPlan{_core.registry, _core.planData, regionId<TRegion>()};	}

	/// @brief Succeed a plan task for a state
	/// @param `stateId` State identifier
	/// @see `HFSM2_ENABLE_PLANS`
	HFSM2_CONSTEXPR(14) void succeed(const StateID stateId_)									noexcept;

	/// @brief Succeed a plan task for a state
	/// @tparam `TState` State type
	/// @see `HFSM2_ENABLE_PLANS`
	template <typename TState>
	HFSM2_CONSTEXPR(14) void succeed()															noexcept	{ succeed(stateId<TState>());							}

	/// @brief Fail a plan task for a state
	/// @param `stateId` State identifier
	/// @see `HFSM2_ENABLE_PLANS`
	HFSM2_CONSTEXPR(14) void fail	(const StateID stateId_)									noexcept;

	/// @brief Fail a plan task for a state
	/// @tparam `TState` State type
	/// @see `HFSM2_ENABLE_PLANS`
	template <typename TState>
	HFSM2_CONSTEXPR(14) void fail	()															noexcept	{ fail	 (stateId<TState>());							}

#endif

	/// @brief Queue a transition into a state (takes effect during `immediate*()`, `update()` or `react()`)
	///   (if transitioning into a region, acts depending on the region type)
	/// @param `stateId` Destination state identifier
	/// @see `immediateChangeTo()`
	HFSM2_CONSTEXPR(14)	void changeTo			(const StateID stateId_)						noexcept;

	/// @brief Queue a transition into a state (takes effect during `immediate*()`, `update()` or `react()`)
	///   (if transitioning into a region, acts depending on the region type)
	/// @tparam `TState` Destination state type
	/// @see `immediateChangeTo()`
	template <typename TState>
	HFSM2_CONSTEXPR(14)	void changeTo			()												noexcept	{ changeTo			(stateId<TState>());				}

	/// @brief Queue a transition into a state (takes effect during `immediate*()`, `update()` or `react()`)
	///   (if transitioning into a region, activates the initial state)
	/// @param `stateId` Destination state identifier
	/// @see `immediateRestart()`
	HFSM2_CONSTEXPR(14)	void restart			(const StateID stateId_)						noexcept;

	/// @brief Transition into a state (if transitioning into a region, activates the initial state)
	/// @tparam `TState` Destination state type
	/// @see `immediateRestart()`
	template <typename TState>
	HFSM2_CONSTEXPR(14)	void restart			()												noexcept	{ restart			(stateId<TState>());				}

	/// @brief Queue a transition into a state (takes effect during `immediate*()`, `update()` or `react()`)
	///   (if transitioning into a region, activates the state that was active previously)
	/// @param `stateId` Destination state identifier
	/// @see `immediateResume()`
	HFSM2_CONSTEXPR(14)	void resume				(const StateID stateId_)						noexcept;

	/// @brief Queue a transition into a state (takes effect during `immediate*()`, `update()` or `react()`)
	///   (if transitioning into a region, activates the state that was active previously)
	/// @tparam `TState` Destination state type
	/// @see `immediateResume()`
	template <typename TState>
	HFSM2_CONSTEXPR(14)	void resume				()												noexcept	{ resume			(stateId<TState>());				}

	/// @brief Queue a transition into a state (takes effect during `immediate*()`, `update()` or `react()`)
	///   (if transitioning into a region, activates the sub-state by index returned by the region's `select()` method)
	/// @param `stateId` Destination state identifier
	/// @see `immediateSelect()`
	HFSM2_CONSTEXPR(14)	void select				(const StateID stateId_)						noexcept;

	/// @brief Queue a transition into a state (takes effect during `immediate*()`, `update()` or `react()`)
	///   (if transitioning into a region, activates the sub-state by index returned by the region's `select()` method)
	/// @tparam `TState` Destination state type
	/// @see `immediateSelect()`
	template <typename TState>
	HFSM2_CONSTEXPR(14)	void select				()												noexcept	{ select			(stateId<TState>());				}

#if HFSM2_UTILITY_THEORY_AVAILABLE()

	/// @brief Queue a transition into a state (takes effect during `immediate*()`, `update()` or `react()`)
	///   (if transitioning into a region, activates the state with the highest `utility()`
	///   among those with the highest `rank()`)
	/// @param `stateId` Destination state identifier
	/// @see `immediateUtilize()`
	/// @see `HFSM2_ENABLE_UTILITY_THEORY`
	HFSM2_CONSTEXPR(14)	void utilize			(const StateID stateId_)						noexcept;

	/// @brief Queue a transition into a state (takes effect during `immediate*()`, `update()` or `react()`)
	///   (if transitioning into a region, activates the state with the highest `utility()`
	///   among those with the highest `rank()`)
	/// @tparam `TState` Destination state type
	/// @see `immediateUtilize()`
	/// @see `HFSM2_ENABLE_UTILITY_THEORY`
	template <typename TState>
	HFSM2_CONSTEXPR(14)	void utilize			()												noexcept	{ utilize			(stateId<TState>());				}

	/// @brief Queue a transition into a state (takes effect during `immediate*()`, `update()` or `react()`)
	///   (if transitioning into a region, uses weighted random to activate the state proportional to `utility()`
	///   among those with the highest `rank()`)
	/// @param `stateId` Destination state identifier
	/// @see `immediateRandomize()`
	/// @see `HFSM2_ENABLE_UTILITY_THEORY`
	HFSM2_CONSTEXPR(14)	void randomize			(const StateID stateId_)						noexcept;

	/// @brief Queue a transition into a state (takes effect during `immediate*()`, `update()` or `react()`)
	///   (if transitioning into a region, uses weighted random to activate the state proportional to `utility()`
	///   among those with the highest `rank()`)
	/// @tparam `TState` Destination state type
	/// @see `immediateSelect()`
	/// @see `HFSM2_ENABLE_UTILITY_THEORY`
	template <typename TState>
	HFSM2_CONSTEXPR(14)	void randomize			()												noexcept	{ randomize			(stateId<TState>());				}

#endif

	/// @brief Schedule a state to be activated when its parent region is activated
	/// @param `stateId` Destination state identifier
	HFSM2_CONSTEXPR(14)	void schedule			(const StateID stateId_)						noexcept;

	/// @brief Schedule a state to be activated when its parent region is activated
	/// @tparam `TState` Destination state type
	template <typename TState>
	HFSM2_CONSTEXPR(14)	void schedule			()												noexcept	{ schedule			(stateId<TState>());				}

	/// @brief Transition into a state
	///   (if transitioning into a region, acts depending on the region type)
	/// @param `stateId` Destination state identifier
	/// @see `changeTo()`
	HFSM2_CONSTEXPR(14)	void immediateChangeTo	(const StateID stateId_)						noexcept;

	/// @brief Transition into a state
	///   (if transitioning into a region, acts depending on the region type)
	/// @tparam `TState` Destination state type
	/// @see `changeTo()`
	template <typename TState>
	HFSM2_CONSTEXPR(14)	void immediateChangeTo	()												noexcept	{ immediateChangeTo	(stateId<TState>());				}

	/// @brief Transition into a state
	///   (if transitioning into a region, activates the initial state)
	/// @param `stateId` Destination state identifier
	/// @see `restart()`
	HFSM2_CONSTEXPR(14)	void immediateRestart	(const StateID stateId_)						noexcept;

	/// @brief Transition into a state (if transitioning into a region, activates the initial state)
	/// @tparam `TState` Destination state type
	/// @see `restart()`
	template <typename TState>
	HFSM2_CONSTEXPR(14)	void immediateRestart	()												noexcept	{ immediateRestart	(stateId<TState>());				}

	/// @brief Transition into a state
	///   (if transitioning into a region, activates the state that was active previously)
	/// @param `stateId` Destination state identifier
	/// @see `resume()`
	HFSM2_CONSTEXPR(14)	void immediateResume	(const StateID stateId_)						noexcept;

	/// @brief Transition into a state (if transitioning into a region, activates the state that was active previously)
	/// @tparam `TState` Destination state type
	/// @see `resume()`
	template <typename TState>
	HFSM2_CONSTEXPR(14)	void immediateResume	()												noexcept	{ immediateResume	(stateId<TState>());				}

	/// @brief Transition into a state
	///   (if transitioning into a region, activates the sub-state by index returned by the region's `select()` method)
	/// @param `stateId` Destination state identifier
	/// @see `select()`
	HFSM2_CONSTEXPR(14)	void immediateSelect	(const StateID stateId_)						noexcept;

	/// @brief Transition into a state
	///   (if transitioning into a region, activates the sub-state by index returned by the region's `select()` method)
	/// @tparam `TState` Destination state type
	/// @see `select()`
	template <typename TState>
	HFSM2_CONSTEXPR(14)	void immediateSelect	()												noexcept	{ immediateSelect	(stateId<TState>());				}

#if HFSM2_UTILITY_THEORY_AVAILABLE()

	/// @brief Transition into a state
	///   (if transitioning into a region, activates the state with the highest `utility()`
	///   among those with the highest `rank()`)
	/// @param `stateId` Destination state identifier
	/// @see `utilize()`
	/// @see `HFSM2_ENABLE_UTILITY_THEORY`
	HFSM2_CONSTEXPR(14)	void immediateUtilize	(const StateID stateId_)						noexcept;

	/// @brief Transition into a state
	///   (if transitioning into a region, activates the state with the highest `utility()`
	///   among those with the highest `rank()`)
	/// @tparam `TState` Destination state type
	/// @see `utilize()`
	/// @see `HFSM2_ENABLE_UTILITY_THEORY`
	template <typename TState>
	HFSM2_CONSTEXPR(14)	void immediateUtilize	()												noexcept	{ immediateUtilize	(stateId<TState>());				}

	/// @brief Transition into a state
	///   (if transitioning into a region, uses weighted random to activate the state proportional to `utility()`
	///   among those with the highest `rank()`)
	/// @param `stateId` Destination state identifier
	/// @see `randomize()`
	/// @see `HFSM2_ENABLE_UTILITY_THEORY`
	HFSM2_CONSTEXPR(14)	void immediateRandomize	(const StateID stateId_)						noexcept;

	/// @brief Transition into a state
	///   (if transitioning into a region, uses weighted random to activate the state proportional to `utility()`
	///   among those with the highest `rank()`)
	/// @tparam `TState` Destination state type
	/// @see `randomize()`
	/// @see `HFSM2_ENABLE_UTILITY_THEORY`
	template <typename TState>
	HFSM2_CONSTEXPR(14)	void immediateRandomize	()												noexcept	{ immediateRandomize(stateId<TState>());				}

#endif

	/// @brief Check if a state is going to be activated or deactivated
	/// @param `stateId` Destination state identifier
	/// @return State pending activation/deactivation status
	HFSM2_CONSTEXPR(11)	bool isPendingChange	(const StateID stateId_)				  const noexcept	{ return _core.registry.isPendingChange(stateId_);		}

	/// @brief Check if a state is going to be activated or deactivated
	/// @tparam `TState` Destination state type
	/// @return State pending activation/deactivation status
	template <typename TState>
	HFSM2_CONSTEXPR(11)	bool isPendingChange	()										  const noexcept	{ return isPendingChange(stateId<TState>());			}

	/// @brief Check if a state is going to be activated
	/// @param `stateId` Destination state identifier
	/// @return State pending activation status
	HFSM2_CONSTEXPR(11)	bool isPendingEnter		(const StateID stateId_)				  const noexcept	{ return _core.registry.isPendingEnter (stateId_);		}

	/// @brief Check if a state is going to be activated
	/// @tparam `TState` Destination state type
	/// @return State pending activation status
	template <typename TState>
	HFSM2_CONSTEXPR(11)	bool isPendingEnter		()										  const noexcept	{ return isPendingEnter (stateId<TState>());			}

	/// @brief Check if a state is going to be deactivated
	/// @param `stateId` Destination state identifier
	/// @return State pending deactivation status
	HFSM2_CONSTEXPR(11)	bool isPendingExit		(const StateID stateId_)				  const noexcept	{ return _core.registry.isPendingExit  (stateId_);		}

	/// @brief Check if a state is going to be deactivated
	/// @tparam `TState` Destination state type
	/// @return State pending deactivation status
	template <typename TState>
	HFSM2_CONSTEXPR(11)	bool isPendingExit		()										  const noexcept	{ return isPendingExit  (stateId<TState>());			}

	/// @brief Reset FSM to initial state (recursively 'exit()' currently active states 'enter()' initial states)
	HFSM2_CONSTEXPR(14)	void reset()															noexcept;

#if HFSM2_STRUCTURE_REPORT_AVAILABLE()

	/// @brief Array of 'StructureEntry' representing FSM structure
	/// @see HFSM2_ENABLE_STRUCTURE_REPORT
	using Structure				= DynamicArrayT<StructureEntry, NAME_COUNT>;

	/// @brief Array of 'int8_t' representing FSM activation history (negative - 'update()' cycles since deactivated, positive - 'update()' cycles since activated)
	/// @see `HFSM2_ENABLE_STRUCTURE_REPORT`
using ActivityHistory		= DynamicArrayT<int8_t,		 NAME_COUNT>;

	/// @brief Get the array of `StructureEntry` representing FSM structure
	/// @return FSM structure
	/// @see `HFSM2_ENABLE_STRUCTURE_REPORT`
	HFSM2_CONSTEXPR(11)	const Structure&	   structure()								  const noexcept	{ return _structure;									}

	/// @brief Get the array of `int8_t` representing FSM activation history (negative - `update()` cycles since deactivated, positive - `update()` cycles since activated)
	/// @return FSM activation history
	/// @see `HFSM2_ENABLE_STRUCTURE_REPORT`
	HFSM2_CONSTEXPR(11)	const ActivityHistory& activityHistory()						  const noexcept	{ return _activityHistory;								}

#endif

#if HFSM2_TRANSITION_HISTORY_AVAILABLE()

	/// @brief Get the transition recorded during last `update()` / `react()`
	/// @return Array of last recorded transitions
	/// @see `HFSM2_ENABLE_TRANSITION_HISTORY`
	HFSM2_CONSTEXPR(11)	const TransitionSets& previousTransitions()						  const noexcept	{ return _core.previousTransitions;						}

	/// @brief Force process transitions (skips `guard()` calls)
	///   Can be used to synchronize multiple FSMs
	/// @param `transitions` Array of 'Transition' to replay
	/// @param `count` Number of transitions
	/// @return Success status
	/// @see `HFSM2_ENABLE_TRANSITION_HISTORY`
	HFSM2_CONSTEXPR(14)	bool replayTransitions(const Transition* const transitions,
											   const Short count)								noexcept;

	/// @brief Force process transitions (skips `guard()` calls)
	///   Can be used to synchronize multiple FSMs
	/// @param `transitions` Array of 'Transition' to replay
	/// @return Success status
	/// @see `HFSM2_ENABLE_TRANSITION_HISTORY`
	template <Long NCount>
	HFSM2_CONSTEXPR(14)	bool replayTransitions(const DynamicArrayT<Transition, NCount>& transitions)	noexcept;

	/// @brief Force process a transition (skips `guard()` calls)
	///   Can be used to synchronize multiple FSMs
	/// @param `transition` 'Transition' to replay
	/// @return Success status
	/// @see `HFSM2_ENABLE_TRANSITION_HISTORY`
	HFSM2_CONSTEXPR(14)	bool replayTransition (const Transition& transition)					noexcept	{ return replayTransitions(&transition, 1);				}

	/// @brief Get the last transition that caused the state to be activated
	/// @param `stateId` State identifier
	/// @return Pointer to the last transition that activated the state
	HFSM2_CONSTEXPR(14)	const Transition* lastTransitionTo(const StateID stateId_)		  const noexcept;

	/// @brief Get the last transition that caused the state to be activated
	/// @tparam `TState` State type
	/// @return Pointer to the last transition that activated the state
	template <typename TState>
	HFSM2_CONSTEXPR(14)	const Transition* lastTransitionTo()							  const noexcept	{ return lastTransitionTo(stateId<TState>());			}

#endif

#if HFSM2_LOG_INTERFACE_AVAILABLE()

	/// @brief Attach logger
	/// @param `logger` A logger implementing 'hfsm2::LoggerInterfaceT<>' interface
	/// @see `HFSM2_ENABLE_LOG_INTERFACE`
	HFSM2_CONSTEXPR(14)	void attachLogger(Logger* const logger)									noexcept	{ _core.logger = logger;								}

#endif

protected:
	HFSM2_CONSTEXPR(14)	void initialEnter()														noexcept;
	HFSM2_CONSTEXPR(14)	void finalExit()														noexcept;

	HFSM2_CONSTEXPR(14)	void processRequest()													noexcept;
	HFSM2_CONSTEXPR(14)	void processTransitions(TransitionSets& currentTransitions)				noexcept;

	HFSM2_CONSTEXPR(14)	bool applyRequests(const TransitionSets& currentTransitions,
										   Control& control)									noexcept;

	HFSM2_CONSTEXPR(14)	bool applyRequest (const TransitionSets& currentTransitions,
										   Control& control,
										   const Transition& request,
										   const Short index)									noexcept;

	HFSM2_CONSTEXPR(14)	bool cancelledByEntryGuards(const TransitionSets& currentTransitions,
													const TransitionSet&  pendingTransitions)	noexcept;

	HFSM2_CONSTEXPR(14)	bool cancelledByGuards(const TransitionSets& currentTransitions,
											   const TransitionSet&  pendingTransitions)		noexcept;

#if HFSM2_SERIALIZATION_AVAILABLE()
	HFSM2_CONSTEXPR(14)	void save(WriteStream& stream)									  const noexcept;
	HFSM2_CONSTEXPR(14)	void load( ReadStream& stream)											noexcept;
#endif

#if HFSM2_TRANSITION_HISTORY_AVAILABLE()
	HFSM2_CONSTEXPR(14)	bool applyRequests(Control& control,
										   const Transition* const transitions,
										   const Short count)									noexcept;
#endif

#if HFSM2_STRUCTURE_REPORT_AVAILABLE()
	HFSM2_CONSTEXPR(14)	void getStateNames()													noexcept;
	HFSM2_CONSTEXPR(14)	void udpateActivity()													noexcept;

Prefixes _prefixes;
NamedStates _namedStates;

Structure _structure;
ActivityHistory _activityHistory;
#endif

protected:
Core _core;
Apex _apex;
};

}
}

namespace hfsm2 {
	namespace detail {

		template <typename TG_, typename TA_>
		HFSM2_CONSTEXPR(14)
		R_<TG_, TA_>::R_(Context& context
		HFSM2_IF_UTILITY_THEORY(, RNG& rng)
		HFSM2_IF_LOG_INTERFACE(, Logger* const logger)) noexcept
		: _core{context
		HFSM2_IF_UTILITY_THEORY(, rng)
	HFSM2_IF_LOG_INTERFACE(, logger)}
	{
	_apex.deepRegister(_core.registry, Parent{});

	HFSM2_IF_STRUCTURE_REPORT(getStateNames());
}

template <typename TG_, typename TA_>
HFSM2_CONSTEXPR(14)
R_<TG_, TA_>::R_(PureContext&& context
			   HFSM2_IF_UTILITY_THEORY(, RNG& rng)
			   HFSM2_IF_LOG_INTERFACE(, Logger* const logger)) noexcept
	: _core{move(context)
		  HFSM2_IF_UTILITY_THEORY(, rng)
		  HFSM2_IF_LOG_INTERFACE(, logger)}
{
_apex.deepRegister(_core.registry, Parent{});

	HFSM2_IF_STRUCTURE_REPORT(getStateNames());
}

template <typename TG_, typename TA_>
HFSM2_CONSTEXPR(20)
R_<TG_, TA_>::~R_() noexcept {
	HFSM2_IF_ASSERT(HFSM2_IF_PLANS(_core.planData.verifyPlans()));
}

template <typename TG_, typename TA_>
HFSM2_CONSTEXPR(14)
void
R_<TG_, TA_>::update() noexcept {
	HFSM2_ASSERT(_core.registry.isActive());

TransitionSets emptyTransitions;
FullControl control{_core, emptyTransitions};

	_apex. deepPreUpdate(control);
	_apex.	  deepUpdate(control);
	_apex.deepPostUpdate(control);

#if HFSM2_PLANS_AVAILABLE()
	_apex.deepUpdatePlans(control);
	_core.planData.clearStatuses();
#endif

	processRequest();
}

template <typename TG_, typename TA_>
template <typename TEvent>
HFSM2_CONSTEXPR(14)
void
R_<TG_, TA_>::react(const TEvent& event) noexcept {
	HFSM2_ASSERT(_core.registry.isActive());

TransitionSets emptyTransitions;
EventControl control{_core, emptyTransitions};

	_apex. deepPreReact(control, event);

control._consumed = false;
	_apex.	  deepReact(control, event);

control._consumed = false;
	_apex.deepPostReact(control, event);

#if HFSM2_PLANS_AVAILABLE()
	_apex.deepUpdatePlans(control);
	_core.planData.clearStatuses();
#endif

	processRequest();
}

template <typename TG_, typename TA_>
template <typename TEvent>
HFSM2_CONSTEXPR(14)
void
R_<TG_, TA_>::query(TEvent& event) const noexcept {
	HFSM2_ASSERT(_core.registry.isActive());

	ConstControl control{_core};

	_apex.deepQuery(control, event);
}

#if HFSM2_PLANS_AVAILABLE()

template <typename TG_, typename TA_>
HFSM2_CONSTEXPR(14)
void
R_<TG_, TA_>::succeed(const StateID stateId_) noexcept {
	if (HFSM2_CHECKED(ROOT_ID < stateId_ && stateId_ < STATE_COUNT)) {
		_core.planData.tasksSuccesses.set(stateId_);

		HFSM2_LOG_TASK_STATUS(_core.context, INVALID_REGION_ID, stateId_, StatusEvent::SUCCEEDED);
	}
}

template <typename TG_, typename TA_>
HFSM2_CONSTEXPR(14)
void
R_<TG_, TA_>::fail(const StateID stateId_) noexcept {
	if (HFSM2_CHECKED(ROOT_ID < stateId_ && stateId_ < STATE_COUNT)) {
		_core.planData.tasksFailures.set(stateId_);

		HFSM2_LOG_TASK_STATUS(_core.context, INVALID_REGION_ID, stateId_, StatusEvent::FAILED);
	}
}

#endif

template <typename TG_, typename TA_>
HFSM2_CONSTEXPR(14)
void
R_<TG_, TA_>::changeTo(const StateID stateId_) noexcept {
	HFSM2_ASSERT(_core.registry.isActive());

_core.requests.emplace(Transition{stateId_, TransitionType::CHANGE});

	HFSM2_LOG_TRANSITION(_core.context, INVALID_STATE_ID, TransitionType::CHANGE, stateId_);
}

template <typename TG_, typename TA_>
HFSM2_CONSTEXPR(14)
void
R_<TG_, TA_>::restart(const StateID stateId_) noexcept {
	HFSM2_ASSERT(_core.registry.isActive());

_core.requests.emplace(Transition{stateId_, TransitionType::RESTART});

	HFSM2_LOG_TRANSITION(_core.context, INVALID_STATE_ID, TransitionType::RESTART, stateId_);
}

template <typename TG_, typename TA_>
HFSM2_CONSTEXPR(14)
void
R_<TG_, TA_>::resume(const StateID stateId_) noexcept {
	HFSM2_ASSERT(_core.registry.isActive());

_core.requests.emplace(Transition{stateId_, TransitionType::RESUME});

	HFSM2_LOG_TRANSITION(_core.context, INVALID_STATE_ID, TransitionType::RESUME, stateId_);
}

template <typename TG_, typename TA_>
HFSM2_CONSTEXPR(14)
void
R_<TG_, TA_>::select(const StateID stateId_) noexcept {
	HFSM2_ASSERT(_core.registry.isActive());

_core.requests.emplace(Transition{stateId_, TransitionType::SELECT});

	HFSM2_LOG_TRANSITION(_core.context, INVALID_STATE_ID, TransitionType::SELECT, stateId_);
}

#if HFSM2_UTILITY_THEORY_AVAILABLE()

template <typename TG_, typename TA_>
HFSM2_CONSTEXPR(14)
void
R_<TG_, TA_>::utilize(const StateID stateId_) noexcept {
	HFSM2_ASSERT(_core.registry.isActive());

_core.requests.emplace(Transition{stateId_, TransitionType::UTILIZE});

	HFSM2_LOG_TRANSITION(_core.context, INVALID_STATE_ID, TransitionType::UTILIZE, stateId_);
}

template <typename TG_, typename TA_>
HFSM2_CONSTEXPR(14)
void
R_<TG_, TA_>::randomize(const StateID stateId_) noexcept {
	HFSM2_ASSERT(_core.registry.isActive());

_core.requests.emplace(Transition{stateId_, TransitionType::RANDOMIZE});

	HFSM2_LOG_TRANSITION(_core.context, INVALID_STATE_ID, TransitionType::RANDOMIZE, stateId_);
}

#endif

template <typename TG_, typename TA_>
HFSM2_CONSTEXPR(14)
void
R_<TG_, TA_>::schedule(const StateID stateId_) noexcept {
	HFSM2_ASSERT(_core.registry.isActive());

_core.requests.emplace(Transition{stateId_, TransitionType::SCHEDULE});

	HFSM2_LOG_TRANSITION(_core.context, INVALID_STATE_ID, TransitionType::SCHEDULE, stateId_);
}

template <typename TG_, typename TA_>
HFSM2_CONSTEXPR(14)
void
R_<TG_, TA_>::immediateChangeTo(const StateID stateId_) noexcept {
	changeTo(stateId_);
```
